LIN {X 0,Y 516.886,Z 94.228,A -85,B 0,C 180,E1 -4924.209,E2 -4924.209} C_VEL
LIN {X 0,Y 516.862,Z 94.224,A -85,B 0,C 180,E1 -4926.776,E2 -4926.776} C_VEL
LIN {X 0,Y 516.942,Z 94.22,A -85,B 0,C 180,E1 -4929.732,E2 -4929.732} C_VEL
LIN {X 0,Y 516.923,Z 94.315,A -85,B 0,C 180,E1 -4932.877,E2 -4932.877} C_VEL
LIN {X 0,Y 518.41,Z 102.009,A -85,B 0,C 180,E1 -4934.268,E2 -4934.268} C_VEL
LIN {X 0,Y 518.118,Z 116.227,A -85,B 0,C 180,E1 -4936.668,E2 -4936.668} C_VEL
LIN {X 0,Y 517.972,Z 120.931,A -85,B 0,C 180,E1 -4937.437,E2 -4937.437} C_VEL
LIN {X 0,Y 520.412,Z 132.652,A -85,B 0,C 180,E1 -4937.694,E2 -4937.694} C_VEL
LIN {X 0,Y 519.711,Z 257.165,A -85,B 0,C 180,E1 -4939.457,E2 -4939.457} C_VEL
LIN {X 0,Y 519.49,Z 271.718,A -85,B 0,C 180,E1 -4939.821,E2 -4939.821} C_VEL
LIN {X 0,Y 519.222,Z 285.007,A -85,B 0,C 180,E1 -4940.308,E2 -4940.308} C_VEL
LIN {X 0,Y 518.835,Z 298.02,A -85,B 0,C 180,E1 -4940.94,E2 -4940.94} C_VEL
LIN {X 0,Y 518.353,Z 311.178,A -85,B 0,C 180,E1 -4941.758,E2 -4941.758} C_VEL
LIN {X 0,Y 517.962,Z 323.367,A -85,B 0,C 180,E1 -4942.706,E2 -4942.706} C_VEL
LIN {X 0,Y 517.606,Z 334.484,A -85,B 0,C 180,E1 -4943.764,E2 -4943.764} C_VEL
LIN {X 0,Y 517.164,Z 344.616,A -85,B 0,C 180,E1 -4944.933,E2 -4944.933} C_VEL
LIN {X 0,Y 516.767,Z 353.015,A -85,B 0,C 180,E1 -4946.101,E2 -4946.101} C_VEL
LIN {X 0,Y 516.612,Z 361.049,A -85,B 0,C 180,E1 -4947.466,E2 -4947.466} C_VEL
LIN {X 0,Y 516.497,Z 367.544,A -85,B 0,C 180,E1 -4948.831,E2 -4948.831} C_VEL
LIN {X 0,Y 516.339,Z 373.334,A -85,B 0,C 180,E1 -4950.39,E2 -4950.39} C_VEL
LIN {X 0,Y 516.219,Z 376.698,A -85,B 0,C 180,E1 -4951.56,E2 -4951.56} C_VEL
LIN {X 0,Y 516.293,Z 379.858,A -85,B 0,C 180,E1 -4953.121,E2 -4953.121} C_VEL
LIN {X 0,Y 516.216,Z 381.664,A -85,B 0,C 180,E1 -4954.686,E2 -4954.686} C_VEL
LIN {X 0,Y 516.295,Z 382.143,A -85,B 0,C 180,E1 -4956.252,E2 -4956.252} C_VEL
LIN {X 0,Y 516.227,Z 381.298,A -85,B 0,C 180,E1 -4957.825,E2 -4957.825} C_VEL
LIN {X 0,Y 516.2,Z 379.096,A -85,B 0,C 180,E1 -4959.403,E2 -4959.403} C_VEL
LIN {X 0,Y 516.363,Z 375.472,A -85,B 0,C 180,E1 -4960.985,E2 -4960.985} C_VEL
LIN {X 0,Y 516.399,Z 370.302,A -85,B 0,C 180,E1 -4962.577,E2 -4962.577} C_VEL
LIN {X 0,Y 516.541,Z 365.25,A -85,B 0,C 180,E1 -4963.775,E2 -4963.775} C_VEL
LIN {X 0,Y 516.733,Z 358.651,A -85,B 0,C 180,E1 -4965.058,E2 -4965.058} C_VEL
LIN {X 0,Y 516.971,Z 350.31,A -85,B 0,C 180,E1 -4966.385,E2 -4966.385} C_VEL
LIN {X 0,Y 517.323,Z 341.381,A -85,B 0,C 180,E1 -4967.554,E2 -4967.554} C_VEL
LIN {X 0,Y 517.693,Z 330.77,A -85,B 0,C 180,E1 -4968.707,E2 -4968.707} C_VEL
LIN {X 0,Y 518.118,Z 319.402,A -85,B 0,C 180,E1 -4969.72,E2 -4969.72} C_VEL
LIN {X 0,Y 518.543,Z 306.72,A -85,B 0,C 180,E1 -4970.633,E2 -4970.633} C_VEL
LIN {X 0,Y 518.93,Z 293.485,A -85,B 0,C 180,E1 -4971.391,E2 -4971.391} C_VEL
LIN {X 0,Y 519.308,Z 279.434,A -85,B 0,C 180,E1 -4972.006,E2 -4972.006} C_VEL
LIN {X 0,Y 519.577,Z 265.737,A -85,B 0,C 180,E1 -4972.439,E2 -4972.439} C_VEL
LIN {X 0,Y 519.75,Z 252.041,A -85,B 0,C 180,E1 -4972.72,E2 -4972.72} C_VEL
LIN {X 0,Y 520.435,Z 132.727,A -85,B 0,C 180,E1 -4974.395,E2 -4974.395} C_VEL
LIN {X 0,Y 517.976,Z 120.735,A -85,B 0,C 180,E1 -4974.681,E2 -4974.681} C_VEL
LIN {X 0,Y 518.432,Z 105.65,A -85,B 0,C 180,E1 -4977.228,E2 -4977.228} C_VEL
LIN {X 0,Y 518.096,Z 100.414,A -85,B 0,C 180,E1 -4978.148,E2 -4978.148} C_VEL
LIN {X 0,Y 516.856,Z 94.228,A -85,B 0,C 180,E1 -4979.309,E2 -4979.309} C_VEL
LIN {X 0,Y 516.865,Z 94.226,A -85,B 0,C 180,E1 -4982.537,E2 -4982.537} C_VEL
LIN {X 0,Y 516.83,Z 94.229,A -85,B 0,C 180,E1 -4985.323,E2 -4985.323} C_VEL
LIN {X 0,Y 516.86,Z 94.224,A -85,B 0,C 180,E1 -4988.718,E2 -4988.718} C_VEL
LIN {X 0,Y 516.832,Z 94.235,A -85,B 0,C 180,E1 -4991.783,E2 -4991.783} C_VEL
LIN {X 0,Y 516.897,Z 94.22,A -85,B 0,C 180,E1 -4995.007,E2 -4995.007} C_VEL
LIN {X 0,Y 516.852,Z 94.225,A -85,B 0,C 180,E1 -4998.407,E2 -4998.407} C_VEL
LIN {X 0,Y 516.872,Z 94.224,A -85,B 0,C 180,E1 -5001.283,E2 -5001.283} C_VEL
LIN {X 0,Y 516.861,Z 94.224,A -85,B 0,C 180,E1 -5004.671,E2 -5004.671} C_VEL
LIN {X 0,Y 516.895,Z 94.223,A -85,B 0,C 180,E1 -5007.457,E2 -5007.457} C_VEL
LIN {X 0,Y 516.904,Z 94.22,A -85,B 0,C 180,E1 -5010.694,E2 -5010.694} C_VEL
LIN {X 0,Y 516.882,Z 94.218,A -85,B 0,C 180,E1 -5013.818,E2 -5013.818} C_VEL
LIN {X 0,Y 516.857,Z 94.23,A -85,B 0,C 180,E1 -5016.776,E2 -5016.776} C_VEL
LIN {X 0,Y 516.938,Z 94.214,A -85,B 0,C 180,E1 -5019.732,E2 -5019.732} C_VEL
LIN {X 0,Y 516.896,Z 94.224,A -85,B 0,C 180,E1 -5022.595,E2 -5022.595} C_VEL
LIN {X 0,Y 516.932,Z 94.215,A -85,B 0,C 180,E1 -5025.03,E2 -5025.03} C_VEL
LIN {X 0,Y 516.967,Z 94.215,A -85,B 0,C 180,E1 -5028.234,E2 -5028.234} C_VEL
LIN {X 0,Y 516.956,Z 94.208,A -85,B 0,C 180,E1 -5031.399,E2 -5031.399} C_VEL
LIN {X 0,Y 517.021,Z 94.205,A -85,B 0,C 180,E1 -5034.54,E2 -5034.54} C_VEL
LIN {X 0,Y 517.081,Z 94.198,A -85,B 0,C 180,E1 -5037.663,E2 -5037.663} C_VEL
LIN {X 0,Y 517.091,Z 94.192,A -85,B 0,C 180,E1 -5040.779,E2 -5040.779} C_VEL
LIN {X 0,Y 516.984,Z 94.208,A -85,B 0,C 180,E1 -5043.117,E2 -5043.117} C_VEL
LIN {X 0,Y 516.977,Z 94.207,A -85,B 0,C 180,E1 -5046.243,E2 -5046.243} C_VEL
LIN {X 0,Y 516.943,Z 94.219,A -85,B 0,C 180,E1 -5049.389,E2 -5049.389} C_VEL
LIN {X 0,Y 516.953,Z 94.215,A -85,B 0,C 180,E1 -5051.807,E2 -5051.807} C_VEL
LIN {X 0,Y 516.944,Z 94.218,A -85,B 0,C 180,E1 -5055.146,E2 -5055.146} C_VEL
LIN {X 0,Y 516.925,Z 94.215,A -85,B 0,C 180,E1 -5058.222,E2 -5058.222} C_VEL
LIN {X 0,Y 516.913,Z 94.217,A -85,B 0,C 180,E1 -5060.701,E2 -5060.701} C_VEL
LIN {X 0,Y 516.903,Z 94.216,A -85,B 0,C 180,E1 -5064.072,E2 -5064.072} C_VEL
LIN {X 0,Y 516.925,Z 94.218,A -85,B 0,C 180,E1 -5066.658,E2 -5066.658} C_VEL
LIN {X 0,Y 516.912,Z 94.217,A -85,B 0,C 180,E1 -5069.524,E2 -5069.524} C_VEL
LIN {X 0,Y 516.899,Z 94.223,A -85,B 0,C 180,E1 -5072.544,E2 -5072.544} C_VEL
LIN {X 0,Y 516.87,Z 94.221,A -85,B 0,C 180,E1 -5075.33,E2 -5075.33} C_VEL
LIN {X 0,Y 516.881,Z 94.222,A -85,B 0,C 180,E1 -5077.943,E2 -5077.943} C_VEL
LIN {X 0,Y 516.885,Z 94.224,A -85,B 0,C 180,E1 -5080.742,E2 -5080.742} C_VEL
LIN {X 0,Y 516.885,Z 94.222,A -85,B 0,C 180,E1 -5082.831,E2 -5082.831} C_VEL
LIN {X 0,Y 516.883,Z 94.225,A -85,B 0,C 180,E1 -5086.097,E2 -5086.097} C_VEL
LIN {X 0,Y 516.916,Z 94.222,A -85,B 0,C 180,E1 -5088.399,E2 -5088.399} C_VEL
LIN {X 0,Y 516.884,Z 94.22,A -85,B 0,C 180,E1 -5091.284,E2 -5091.284} C_VEL
LIN {X 0,Y 516.872,Z 94.226,A -85,B 0,C 180,E1 -5094.22,E2 -5094.22} C_VEL
LIN {X 0,Y 516.896,Z 94.217,A -85,B 0,C 180,E1 -5097.053,E2 -5097.053} C_VEL
LIN {X 0,Y 516.893,Z 94.226,A -85,B 0,C 180,E1 -5099.796,E2 -5099.796} C_VEL
LIN {X 0,Y 516.93,Z 94.219,A -85,B 0,C 180,E1 -5102.467,E2 -5102.467} C_VEL
LIN {X 0,Y 516.957,Z 94.246,A -85,B 0,C 180,E1 -5104.047,E2 -5104.047} C_VEL
LIN {X 0,Y 518.949,Z 103.849,A -85,B 0,C 180,E1 -5105.633,E2 -5105.633} C_VEL
LIN {X 0,Y 518.879,Z 112.01,A -85,B 0,C 180,E1 -5106.872,E2 -5106.872} C_VEL
LIN {X 0,Y 518.251,Z 131.547,A -85,B 0,C 180,E1 -5109.769,E2 -5109.769} C_VEL
LIN {X 0,Y 517.976,Z 142.613,A -85,B 0,C 180,E1 -5111.377,E2 -5111.377} C_VEL
LIN {X 0,Y 520.411,Z 156.781,A -85,B 0,C 180,E1 -5111.67,E2 -5111.67} C_VEL
LIN {X 0,Y 519.606,Z 280.718,A -85,B 0,C 180,E1 -5113.423,E2 -5113.423} C_VEL
LIN {X 0,Y 519.341,Z 295.01,A -85,B 0,C 180,E1 -5113.785,E2 -5113.785} C_VEL
LIN {X 0,Y 519.059,Z 308.626,A -85,B 0,C 180,E1 -5114.288,E2 -5114.288} C_VEL
LIN {X 0,Y 518.678,Z 320.831,A -85,B 0,C 180,E1 -5114.88,E2 -5114.88} C_VEL
LIN {X 0,Y 518.212,Z 333.672,A -85,B 0,C 180,E1 -5115.67,E2 -5115.67} C_VEL
LIN {X 0,Y 517.839,Z 345.351,A -85,B 0,C 180,E1 -5116.56,E2 -5116.56} C_VEL
LIN {X 0,Y 517.487,Z 355.071,A -85,B 0,C 180,E1 -5117.45,E2 -5117.45} C_VEL
LIN {X 0,Y 517.156,Z 365.842,A -85,B 0,C 180,E1 -5118.635,E2 -5118.635} C_VEL
LIN {X 0,Y 516.819,Z 374.735,A -85,B 0,C 180,E1 -5119.818,E2 -5119.818} C_VEL
LIN {X 0,Y 516.608,Z 383.26,A -85,B 0,C 180,E1 -5121.196,E2 -5121.196} C_VEL
LIN {X 0,Y 516.441,Z 390.13,A -85,B 0,C 180,E1 -5122.572,E2 -5122.572} C_VEL
LIN {X 0,Y 516.357,Z 394.866,A -85,B 0,C 180,E1 -5123.749,E2 -5123.749} C_VEL
LIN {X 0,Y 516.303,Z 398.702,A -85,B 0,C 180,E1 -5124.924,E2 -5124.924} C_VEL
LIN {X 0,Y 516.324,Z 401.659,A -85,B 0,C 180,E1 -5126.097,E2 -5126.097} C_VEL
LIN {X 0,Y 516.259,Z 404.364,A -85,B 0,C 180,E1 -5127.659,E2 -5127.659} C_VEL
LIN {X 0,Y 516.156,Z 405.704,A -85,B 0,C 180,E1 -5129.22,E2 -5129.22} C_VEL
LIN {X 0,Y 516.156,Z 405.706,A -85,B 0,C 180,E1 -5130.78,E2 -5130.78} C_VEL
LIN {X 0,Y 516.259,Z 404.371,A -85,B 0,C 180,E1 -5132.34,E2 -5132.34} C_VEL
LIN {X 0,Y 516.324,Z 401.67,A -85,B 0,C 180,E1 -5133.902,E2 -5133.902} C_VEL
LIN {X 0,Y 516.353,Z 397.525,A -85,B 0,C 180,E1 -5135.467,E2 -5135.467} C_VEL
LIN {X 0,Y 516.4,Z 391.816,A -85,B 0,C 180,E1 -5137.035,E2 -5137.035} C_VEL
LIN {X 0,Y 516.565,Z 385.381,A -85,B 0,C 180,E1 -5138.41,E2 -5138.41} C_VEL
LIN {X 0,Y 516.753,Z 377.385,A -85,B 0,C 180,E1 -5139.788,E2 -5139.788} C_VEL
LIN {X 0,Y 517.059,Z 369.025,A -85,B 0,C 180,E1 -5140.97,E2 -5140.97} C_VEL
LIN {X 0,Y 517.408,Z 358.729,A -85,B 0,C 180,E1 -5142.179,E2 -5142.179} C_VEL
LIN {X 0,Y 517.77,Z 347.731,A -85,B 0,C 180,E1 -5143.241,E2 -5143.241} C_VEL
LIN {X 0,Y 518.118,Z 336.563,A -85,B 0,C 180,E1 -5144.132,E2 -5144.132} C_VEL
LIN {X 0,Y 518.536,Z 324.404,A -85,B 0,C 180,E1 -5144.923,E2 -5144.923} C_VEL
LIN {X 0,Y 518.993,Z 310.915,A -85,B 0,C 180,E1 -5145.613,E2 -5145.613} C_VEL
LIN {X 0,Y 519.284,Z 296.756,A -85,B 0,C 180,E1 -5146.16,E2 -5146.16} C_VEL
LIN {X 0,Y 519.595,Z 281.901,A -85,B 0,C 180,E1 -5146.552,E2 -5146.552} C_VEL
LIN {X 0,Y 519.83,Z 251.984,A -85,B 0,C 180,E1 -5146.999,E2 -5146.999} C_VEL
LIN {X 0,Y 520.344,Z 155.931,A -85,B 0,C 180,E1 -5148.345,E2 -5148.345} C_VEL
LIN {X 0,Y 517.993,Z 142.476,A -85,B 0,C 180,E1 -5148.634,E2 -5148.634} C_VEL
LIN {X 0,Y 518.563,Z 120.29,A -85,B 0,C 180,E1 -5151.882,E2 -5151.882} C_VEL
LIN {X 0,Y 519.05,Z 104.898,A -85,B 0,C 180,E1 -5154.163,E2 -5154.163} C_VEL
LIN {X 0,Y 516.961,Z 94.218,A -85,B 0,C 180,E1 -5155.889,E2 -5155.889} C_VEL
LIN {X 0,Y 516.92,Z 94.222,A -85,B 0,C 180,E1 -5158.415,E2 -5158.415} C_VEL
LIN {X 0,Y 516.889,Z 94.221,A -85,B 0,C 180,E1 -5161.109,E2 -5161.109} C_VEL
LIN {X 0,Y 516.908,Z 94.223,A -85,B 0,C 180,E1 -5163.966,E2 -5163.966} C_VEL
LIN {X 0,Y 516.876,Z 94.222,A -85,B 0,C 180,E1 -5166.746,E2 -5166.746} C_VEL
LIN {X 0,Y 516.882,Z 94.225,A -85,B 0,C 180,E1 -5169.721,E2 -5169.721} C_VEL
LIN {X 0,Y 516.914,Z 94.223,A -85,B 0,C 180,E1 -5171.775,E2 -5171.775} C_VEL
LIN {X 0,Y 516.922,Z 94.215,A -85,B 0,C 180,E1 -5175.01,E2 -5175.01} C_VEL
LIN {X 0,Y 516.915,Z 94.217,A -85,B 0,C 180,E1 -5178.398,E2 -5178.398} C_VEL
LIN {X 0,Y 516.879,Z 94.225,A -85,B 0,C 180,E1 -5181.284,E2 -5181.284} C_VEL
LIN {X 0,Y 516.87,Z 94.222,A -85,B 0,C 180,E1 -5184.22,E2 -5184.22} C_VEL
LIN {X 0,Y 516.895,Z 94.222,A -85,B 0,C 180,E1 -5187.053,E2 -5187.053} C_VEL
LIN {X 0,Y 516.891,Z 94.221,A -85,B 0,C 180,E1 -5189.796,E2 -5189.796} C_VEL
LIN {X 0,Y 516.925,Z 94.215,A -85,B 0,C 180,E1 -5192.467,E2 -5192.467} C_VEL
LIN {X 0,Y 516.908,Z 94.225,A -85,B 0,C 180,E1 -5195.072,E2 -5195.072} C_VEL
LIN {X 0,Y 516.884,Z 94.222,A -85,B 0,C 180,E1 -5198.462,E2 -5198.462} C_VEL
LIN {X 0,Y 516.901,Z 94.227,A -85,B 0,C 180,E1 -5200.955,E2 -5200.955} C_VEL
LIN {X 0,Y 516.912,Z 94.218,A -85,B 0,C 180,E1 -5203.41,E2 -5203.41} C_VEL
LIN {X 0,Y 516.895,Z 94.218,A -85,B 0,C 180,E1 -5205.834,E2 -5205.834} C_VEL
LIN {X 0,Y 516.965,Z 94.212,A -85,B 0,C 180,E1 -5208.234,E2 -5208.234} C_VEL
LIN {X 0,Y 516.967,Z 94.21,A -85,B 0,C 180,E1 -5211.4,E2 -5211.4} C_VEL
LIN {X 0,Y 517.008,Z 94.205,A -85,B 0,C 180,E1 -5213.757,E2 -5213.757} C_VEL
LIN {X 0,Y 517.082,Z 94.196,A -85,B 0,C 180,E1 -5217.663,E2 -5217.663} C_VEL
LIN {X 0,Y 517.092,Z 94.196,A -85,B 0,C 180,E1 -5220.779,E2 -5220.779} C_VEL
LIN {X 0,Y 517.011,Z 94.204,A -85,B 0,C 180,E1 -5223.117,E2 -5223.117} C_VEL
LIN {X 0,Y 516.988,Z 94.214,A -85,B 0,C 180,E1 -5226.244,E2 -5226.244} C_VEL
LIN {X 0,Y 516.968,Z 94.211,A -85,B 0,C 180,E1 -5228.601,E2 -5228.601} C_VEL
LIN {X 0,Y 516.952,Z 94.219,A -85,B 0,C 180,E1 -5231.807,E2 -5231.807} C_VEL
LIN {X 0,Y 516.944,Z 94.213,A -85,B 0,C 180,E1 -5235.147,E2 -5235.147} C_VEL
LIN {X 0,Y 516.912,Z 94.218,A -85,B 0,C 180,E1 -5238.223,E2 -5238.223} C_VEL
LIN {X 0,Y 516.912,Z 94.216,A -85,B 0,C 180,E1 -5240.702,E2 -5240.702} C_VEL
LIN {X 0,Y 516.891,Z 94.221,A -85,B 0,C 180,E1 -5244.073,E2 -5244.073} C_VEL
LIN {X 0,Y 516.925,Z 94.215,A -85,B 0,C 180,E1 -5246.658,E2 -5246.658} C_VEL
LIN {X 0,Y 516.908,Z 94.223,A -85,B 0,C 180,E1 -5249.524,E2 -5249.524} C_VEL
LIN {X 0,Y 516.894,Z 94.219,A -85,B 0,C 180,E1 -5252.543,E2 -5252.543} C_VEL
LIN {X 0,Y 516.865,Z 94.228,A -85,B 0,C 180,E1 -5255.33,E2 -5255.33} C_VEL
LIN {X 0,Y 516.879,Z 94.22,A -85,B 0,C 180,E1 -5257.943,E2 -5257.943} C_VEL
LIN {X 0,Y 516.883,Z 94.225,A -85,B 0,C 180,E1 -5260.742,E2 -5260.742} C_VEL
LIN {X 0,Y 516.883,Z 94.228,A -85,B 0,C 180,E1 -5262.832,E2 -5262.832} C_VEL
LIN {X 0,Y 516.896,Z 94.224,A -85,B 0,C 180,E1 -5265.007,E2 -5265.007} C_VEL
LIN {X 0,Y 516.911,Z 94.221,A -85,B 0,C 180,E1 -5268.4,E2 -5268.4} C_VEL
LIN {X 0,Y 516.882,Z 94.224,A -85,B 0,C 180,E1 -5270.287,E2 -5270.287} C_VEL
LIN {X 0,Y 516.207,Z 94.309,A -85,B 0,C 180,E1 -5270.937,E2 -5270.937} C_VEL
LIN {X 0,Y 513.349,Z 94.662,A -85,B 0,C 180,E1 -5271.993,E2 -5271.993} C_VEL
LIN {X 0,Y 510.935,Z 94.966,A -85,B 0,C 180,E1 -5272.843,E2 -5272.843} C_VEL
LIN {X 0,Y 509.895,Z 95.091,A -85,B 0,C 180,E1 -5273.499,E2 -5273.499} C_VEL
LIN {X 0,Y 509.808,Z 95.102,A -85,B 0,C 180,E1 -5273.722,E2 -5273.722} C_VEL
LIN {X 0,Y 509.86,Z 95.102,A -85,B 0,C 180,E1 -5276.539,E2 -5276.539} C_VEL
LIN {X 0,Y 509.847,Z 95.096,A -85,B 0,C 180,E1 -5279.335,E2 -5279.335} C_VEL
LIN {X 0,Y 509.847,Z 95.102,A -85,B 0,C 180,E1 -5282.052,E2 -5282.052} C_VEL
LIN {X 0,Y 509.817,Z 95.102,A -85,B 0,C 180,E1 -5284.701,E2 -5284.701} C_VEL
LIN {X 0,Y 509.829,Z 95.1,A -85,B 0,C 180,E1 -5287.458,E2 -5287.458} C_VEL
LIN {X 0,Y 509.919,Z 95.096,A -85,B 0,C 180,E1 -5289.845,E2 -5289.845} C_VEL
LIN {X 0,Y 509.892,Z 95.19,A -85,B 0,C 180,E1 -5292.685,E2 -5292.685} C_VEL
LIN {X 0,Y 511.532,Z 104.027,A -85,B 0,C 180,E1 -5294.299,E2 -5294.299} C_VEL
LIN {X 0,Y 511.03,Z 120.993,A -85,B 0,C 180,E1 -5297.18,E2 -5297.18} C_VEL
LIN {X 0,Y 513.74,Z 134.085,A -85,B 0,C 180,E1 -5297.47,E2 -5297.47} C_VEL
LIN {X 0,Y 512.923,Z 257.73,A -85,B 0,C 180,E1 -5299.241,E2 -5299.241} C_VEL
LIN {X 0,Y 512.673,Z 272.139,A -85,B 0,C 180,E1 -5299.61,E2 -5299.61} C_VEL
LIN {X 0,Y 512.372,Z 285.921,A -85,B 0,C 180,E1 -5300.128,E2 -5300.128} C_VEL
LIN {X 0,Y 511.921,Z 299.648,A -85,B 0,C 180,E1 -5300.817,E2 -5300.817} C_VEL
LIN {X 0,Y 511.442,Z 312.046,A -85,B 0,C 180,E1 -5301.611,E2 -5301.611} C_VEL
LIN {X 0,Y 511.025,Z 324.435,A -85,B 0,C 180,E1 -5302.6,E2 -5302.6} C_VEL
LIN {X 0,Y 510.626,Z 335.443,A -85,B 0,C 180,E1 -5303.679,E2 -5303.679} C_VEL
LIN {X 0,Y 510.151,Z 345.407,A -85,B 0,C 180,E1 -5304.863,E2 -5304.863} C_VEL
LIN {X 0,Y 509.725,Z 353.706,A -85,B 0,C 180,E1 -5306.047,E2 -5306.047} C_VEL
LIN {X 0,Y 509.557,Z 361.633,A -85,B 0,C 180,E1 -5307.431,E2 -5307.431} C_VEL
LIN {X 0,Y 509.413,Z 368.046,A -85,B 0,C 180,E1 -5308.814,E2 -5308.814} C_VEL
LIN {X 0,Y 509.262,Z 373.758,A -85,B 0,C 180,E1 -5310.395,E2 -5310.395} C_VEL
LIN {X 0,Y 509.138,Z 377.054,A -85,B 0,C 180,E1 -5311.582,E2 -5311.582} C_VEL
LIN {X 0,Y 509.207,Z 380.139,A -85,B 0,C 180,E1 -5313.165,E2 -5313.165} C_VEL
LIN {X 0,Y 509.131,Z 381.877,A -85,B 0,C 180,E1 -5314.751,E2 -5314.751} C_VEL
LIN {X 0,Y 509.221,Z 382.271,A -85,B 0,C 180,E1 -5316.429,E2 -5316.429} C_VEL
LIN {X 0,Y 509.142,Z 381.376,A -85,B 0,C 180,E1 -5317.934,E2 -5317.934} C_VEL
LIN {X 0,Y 509.114,Z 379.104,A -85,B 0,C 180,E1 -5319.535,E2 -5319.535} C_VEL
LIN {X 0,Y 509.298,Z 375.407,A -85,B 0,C 180,E1 -5321.139,E2 -5321.139} C_VEL
LIN {X 0,Y 509.363,Z 370.155,A -85,B 0,C 180,E1 -5322.754,E2 -5322.754} C_VEL
LIN {X 0,Y 509.495,Z 365.022,A -85,B 0,C 180,E1 -5323.969,E2 -5323.969} C_VEL
LIN {X 0,Y 509.754,Z 357.657,A -85,B 0,C 180,E1 -5325.391,E2 -5325.391} C_VEL
LIN {X 0,Y 510.054,Z 348.445,A -85,B 0,C 180,E1 -5326.82,E2 -5326.82} C_VEL
LIN {X 0,Y 510.414,Z 338.458,A -85,B 0,C 180,E1 -5328.077,E2 -5328.077} C_VEL
LIN {X 0,Y 510.865,Z 327.876,A -85,B 0,C 180,E1 -5329.175,E2 -5329.175} C_VEL
LIN {X 0,Y 511.32,Z 315.823,A -85,B 0,C 180,E1 -5330.201,E2 -5330.201} C_VEL
LIN {X 0,Y 511.771,Z 304.056,A -85,B 0,C 180,E1 -5331.014,E2 -5331.014} C_VEL
LIN {X 0,Y 512.189,Z 291.84,A -85,B 0,C 180,E1 -5331.692,E2 -5331.692} C_VEL
LIN {X 0,Y 512.525,Z 278.694,A -85,B 0,C 180,E1 -5332.26,E2 -5332.26} C_VEL
LIN {X 0,Y 512.776,Z 264.818,A -85,B 0,C 180,E1 -5332.695,E2 -5332.695} C_VEL
LIN {X 0,Y 512.975,Z 251.108,A -85,B 0,C 180,E1 -5332.967,E2 -5332.967} C_VEL
LIN {X 0,Y 513.774,Z 134.042,A -85,B 0,C 180,E1 -5334.631,E2 -5334.631} C_VEL
LIN {X 0,Y 511.065,Z 120.93,A -85,B 0,C 180,E1 -5334.944,E2 -5334.944} C_VEL
LIN {X 0,Y 511.57,Z 105.313,A -85,B 0,C 180,E1 -5337.624,E2 -5337.624} C_VEL
LIN {X 0,Y 510.327,Z 97.623,A -85,B 0,C 180,E1 -5339.042,E2 -5339.042} C_VEL
LIN {X 0,Y 509.808,Z 95.107,A -85,B 0,C 180,E1 -5339.538,E2 -5339.538} C_VEL
LIN {X 0,Y 509.833,Z 95.103,A -85,B 0,C 180,E1 -5342.521,E2 -5342.521} C_VEL
LIN {X 0,Y 509.791,Z 95.106,A -85,B 0,C 180,E1 -5345.381,E2 -5345.381} C_VEL
LIN {X 0,Y 509.809,Z 95.105,A -85,B 0,C 180,E1 -5348.342,E2 -5348.342} C_VEL
LIN {X 0,Y 509.784,Z 95.111,A -85,B 0,C 180,E1 -5351.433,E2 -5351.433} C_VEL
LIN {X 0,Y 509.836,Z 95.099,A -85,B 0,C 180,E1 -5354.67,E2 -5354.67} C_VEL
LIN {X 0,Y 509.79,Z 95.112,A -85,B 0,C 180,E1 -5357.505,E2 -5357.505} C_VEL
LIN {X 0,Y 509.831,Z 95.094,A -85,B 0,C 180,E1 -5360.646,E2 -5360.646} C_VEL
LIN {X 0,Y 509.804,Z 95.105,A -85,B 0,C 180,E1 -5363.645,E2 -5363.645} C_VEL
LIN {X 0,Y 509.84,Z 95.099,A -85,B 0,C 180,E1 -5366.537,E2 -5366.537} C_VEL
LIN {X 0,Y 509.834,Z 95.102,A -85,B 0,C 180,E1 -5369.333,E2 -5369.333} C_VEL
LIN {X 0,Y 509.834,Z 95.099,A -85,B 0,C 180,E1 -5372.051,E2 -5372.051} C_VEL
LIN {X 0,Y 509.802,Z 95.106,A -85,B 0,C 180,E1 -5374.7,E2 -5374.7} C_VEL
LIN {X 0,Y 509.825,Z 95.098,A -85,B 0,C 180,E1 -5377.459,E2 -5377.459} C_VEL
LIN {X 0,Y 509.916,Z 95.089,A -85,B 0,C 180,E1 -5379.844,E2 -5379.844} C_VEL
LIN {X 0,Y 509.864,Z 95.096,A -85,B 0,C 180,E1 -5383.174,E2 -5383.174} C_VEL
LIN {X 0,Y 509.847,Z 95.096,A -85,B 0,C 180,E1 -5385.633,E2 -5385.633} C_VEL
LIN {X 0,Y 509.913,Z 95.091,A -85,B 0,C 180,E1 -5388.874,E2 -5388.874} C_VEL
LIN {X 0,Y 509.922,Z 95.09,A -85,B 0,C 180,E1 -5392.078,E2 -5392.078} C_VEL
LIN {X 0,Y 509.972,Z 95.084,A -85,B 0,C 180,E1 -5394.464,E2 -5394.464} C_VEL
LIN {X 0,Y 510.051,Z 95.073,A -85,B 0,C 180,E1 -5397.631,E2 -5397.631} C_VEL
LIN {X 0,Y 510.062,Z 95.067,A -85,B 0,C 180,E1 -5400.789,E2 -5400.789} C_VEL
LIN {X 0,Y 509.928,Z 95.087,A -85,B 0,C 180,E1 -5403.16,E2 -5403.16} C_VEL
LIN {X 0,Y 509.924,Z 95.085,A -85,B 0,C 180,E1 -5406.33,E2 -5406.33} C_VEL
LIN {X 0,Y 509.911,Z 95.089,A -85,B 0,C 180,E1 -5408.72,E2 -5408.72} C_VEL
LIN {X 0,Y 509.905,Z 95.091,A -85,B 0,C 180,E1 -5411.932,E2 -5411.932} C_VEL
LIN {X 0,Y 509.895,Z 95.097,A -85,B 0,C 180,E1 -5415.242,E2 -5415.242} C_VEL
LIN {X 0,Y 509.883,Z 95.093,A -85,B 0,C 180,E1 -5417.998,E2 -5417.998} C_VEL
LIN {X 0,Y 509.851,Z 95.099,A -85,B 0,C 180,E1 -5421.002,E2 -5421.002} C_VEL
LIN {X 0,Y 509.865,Z 95.094,A -85,B 0,C 180,E1 -5424.426,E2 -5424.426} C_VEL
LIN {X 0,Y 509.885,Z 95.098,A -85,B 0,C 180,E1 -5427.056,E2 -5427.056} C_VEL
LIN {X 0,Y 509.858,Z 95.095,A -85,B 0,C 180,E1 -5429.751,E2 -5429.751} C_VEL
LIN {X 0,Y 509.876,Z 95.099,A -85,B 0,C 180,E1 -5432.774,E2 -5432.774} C_VEL
LIN {X 0,Y 509.828,Z 95.098,A -85,B 0,C 180,E1 -5435.579,E2 -5435.579} C_VEL
LIN {X 0,Y 509.85,Z 95.103,A -85,B 0,C 180,E1 -5438.338,E2 -5438.338} C_VEL
LIN {X 0,Y 509.857,Z 95.095,A -85,B 0,C 180,E1 -5441.425,E2 -5441.425} C_VEL
LIN {X 0,Y 509.84,Z 95.1,A -85,B 0,C 180,E1 -5444.67,E2 -5444.67} C_VEL
LIN {X 0,Y 509.835,Z 95.1,A -85,B 0,C 180,E1 -5447.51,E2 -5447.51} C_VEL
LIN {X 0,Y 509.848,Z 95.097,A -85,B 0,C 180,E1 -5450.648,E2 -5450.648} C_VEL
LIN {X 0,Y 509.826,Z 95.103,A -85,B 0,C 180,E1 -5453.647,E2 -5453.647} C_VEL
LIN {X 0,Y 509.86,Z 95.093,A -85,B 0,C 180,E1 -5456.539,E2 -5456.539} C_VEL
LIN {X 0,Y 509.847,Z 95.1,A -85,B 0,C 180,E1 -5459.334,E2 -5459.334} C_VEL
LIN {X 0,Y 509.895,Z 95.098,A -85,B 0,C 180,E1 -5462.055,E2 -5462.055} C_VEL
LIN {X 0,Y 509.949,Z 95.299,A -85,B 0,C 180,E1 -5463.831,E2 -5463.831} C_VEL
LIN {X 0,Y 512.172,Z 106.4,A -85,B 0,C 180,E1 -5465.691,E2 -5465.691} C_VEL
LIN {X 0,Y 511.65,Z 123.095,A -85,B 0,C 180,E1 -5468.231,E2 -5468.231} C_VEL
LIN {X 0,Y 511.065,Z 142.619,A -85,B 0,C 180,E1 -5471.112,E2 -5471.112} C_VEL
LIN {X 0,Y 513.686,Z 157.572,A -85,B 0,C 180,E1 -5471.431,E2 -5471.431} C_VEL
LIN {X 0,Y 512.807,Z 280.587,A -85,B 0,C 180,E1 -5473.196,E2 -5473.196} C_VEL
LIN {X 0,Y 512.533,Z 294.614,A -85,B 0,C 180,E1 -5473.555,E2 -5473.555} C_VEL
LIN {X 0,Y 512.202,Z 308.464,A -85,B 0,C 180,E1 -5474.072,E2 -5474.072} C_VEL
LIN {X 0,Y 511.727,Z 322.43,A -85,B 0,C 180,E1 -5474.772,E2 -5474.772} C_VEL
LIN {X 0,Y 511.247,Z 334.93,A -85,B 0,C 180,E1 -5475.572,E2 -5475.572} C_VEL
LIN {X 0,Y 510.847,Z 346.358,A -85,B 0,C 180,E1 -5476.474,E2 -5476.474} C_VEL
LIN {X 0,Y 510.453,Z 356.862,A -85,B 0,C 180,E1 -5477.476,E2 -5477.476} C_VEL
LIN {X 0,Y 510.114,Z 367.308,A -85,B 0,C 180,E1 -5478.678,E2 -5478.678} C_VEL
LIN {X 0,Y 509.758,Z 375.928,A -85,B 0,C 180,E1 -5479.876,E2 -5479.876} C_VEL
LIN {X 0,Y 509.521,Z 384.185,A -85,B 0,C 180,E1 -5481.273,E2 -5481.273} C_VEL
LIN {X 0,Y 509.365,Z 389.964,A -85,B 0,C 180,E1 -5482.468,E2 -5482.468} C_VEL
LIN {X 0,Y 509.263,Z 394.7,A -85,B 0,C 180,E1 -5483.661,E2 -5483.661} C_VEL
LIN {X 0,Y 509.232,Z 398.538,A -85,B 0,C 180,E1 -5484.853,E2 -5484.853} C_VEL
LIN {X 0,Y 509.216,Z 401.494,A -85,B 0,C 180,E1 -5486.043,E2 -5486.043} C_VEL
LIN {X 0,Y 509.188,Z 404.201,A -85,B 0,C 180,E1 -5487.627,E2 -5487.627} C_VEL
LIN {X 0,Y 509.07,Z 405.541,A -85,B 0,C 180,E1 -5489.209,E2 -5489.209} C_VEL
LIN {X 0,Y 509.07,Z 405.543,A -85,B 0,C 180,E1 -5490.791,E2 -5490.791} C_VEL
LIN {X 0,Y 509.188,Z 404.209,A -85,B 0,C 180,E1 -5492.373,E2 -5492.373} C_VEL
LIN {X 0,Y 509.216,Z 401.507,A -85,B 0,C 180,E1 -5493.957,E2 -5493.957} C_VEL
LIN {X 0,Y 509.267,Z 397.362,A -85,B 0,C 180,E1 -5495.543,E2 -5495.543} C_VEL
LIN {X 0,Y 509.325,Z 391.652,A -85,B 0,C 180,E1 -5497.134,E2 -5497.134} C_VEL
LIN {X 0,Y 509.508,Z 385.217,A -85,B 0,C 180,E1 -5498.527,E2 -5498.527} C_VEL
LIN {X 0,Y 509.708,Z 377.221,A -85,B 0,C 180,E1 -5499.925,E2 -5499.925} C_VEL
LIN {X 0,Y 510.036,Z 368.86,A -85,B 0,C 180,E1 -5501.123,E2 -5501.123} C_VEL
LIN {X 0,Y 510.391,Z 358.154,A -85,B 0,C 180,E1 -5502.394,E2 -5502.394} C_VEL
LIN {X 0,Y 510.817,Z 347.565,A -85,B 0,C 180,E1 -5503.425,E2 -5503.425} C_VEL
LIN {X 0,Y 511.204,Z 336.397,A -85,B 0,C 180,E1 -5504.327,E2 -5504.327} C_VEL
LIN {X 0,Y 511.644,Z 324.236,A -85,B 0,C 180,E1 -5505.128,E2 -5505.128} C_VEL
LIN {X 0,Y 512.148,Z 310.745,A -85,B 0,C 180,E1 -5505.827,E2 -5505.827} C_VEL
LIN {X 0,Y 512.46,Z 296.743,A -85,B 0,C 180,E1 -5506.376,E2 -5506.376} C_VEL
LIN {X 0,Y 512.791,Z 282.839,A -85,B 0,C 180,E1 -5506.753,E2 -5506.753} C_VEL
LIN {X 0,Y 513.005,Z 262.477,A -85,B 0,C 180,E1 -5507.079,E2 -5507.079} C_VEL
LIN {X 0,Y 513.559,Z 156.679,A -85,B 0,C 180,E1 -5508.581,E2 -5508.581} C_VEL
LIN {X 0,Y 511.044,Z 142.305,A -85,B 0,C 180,E1 -5508.893,E2 -5508.893} C_VEL
LIN {X 0,Y 511.639,Z 121.473,A -85,B 0,C 180,E1 -5511.982,E2 -5511.982} C_VEL
LIN {X 0,Y 512.11,Z 105.965,A -85,B 0,C 180,E1 -5514.312,E2 -5514.312} C_VEL
LIN {X 0,Y 509.909,Z 95.097,A -85,B 0,C 180,E1 -5516.116,E2 -5516.116} C_VEL
LIN {X 0,Y 509.877,Z 95.098,A -85,B 0,C 180,E1 -5518.844,E2 -5518.844} C_VEL
LIN {X 0,Y 509.82,Z 95.103,A -85,B 0,C 180,E1 -5521.59,E2 -5521.59} C_VEL
LIN {X 0,Y 509.847,Z 95.101,A -85,B 0,C 180,E1 -5524.414,E2 -5524.414} C_VEL
LIN {X 0,Y 509.817,Z 95.101,A -85,B 0,C 180,E1 -5527.341,E2 -5527.341} C_VEL
LIN {X 0,Y 509.838,Z 95.1,A -85,B 0,C 180,E1 -5530.382,E2 -5530.382} C_VEL
LIN {X 0,Y 509.824,Z 95.1,A -85,B 0,C 180,E1 -5533.062,E2 -5533.062} C_VEL
LIN {X 0,Y 509.831,Z 95.107,A -85,B 0,C 180,E1 -5535.792,E2 -5535.792} C_VEL
LIN {X 0,Y 509.856,Z 95.095,A -85,B 0,C 180,E1 -5538.575,E2 -5538.575} C_VEL
LIN {X 0,Y 509.85,Z 95.102,A -85,B 0,C 180,E1 -5541.786,E2 -5541.786} C_VEL
LIN {X 0,Y 509.829,Z 95.099,A -85,B 0,C 180,E1 -5544.622,E2 -5544.622} C_VEL
LIN {X 0,Y 509.862,Z 95.102,A -85,B 0,C 180,E1 -5547.481,E2 -5547.481} C_VEL
LIN {X 0,Y 509.857,Z 95.095,A -85,B 0,C 180,E1 -5550.274,E2 -5550.274} C_VEL
LIN {X 0,Y 509.883,Z 95.097,A -85,B 0,C 180,E1 -5552.944,E2 -5552.944} C_VEL
LIN {X 0,Y 509.864,Z 95.097,A -85,B 0,C 180,E1 -5555.574,E2 -5555.574} C_VEL
LIN {X 0,Y 509.849,Z 95.105,A -85,B 0,C 180,E1 -5558.998,E2 -5558.998} C_VEL
LIN {X 0,Y 509.881,Z 95.092,A -85,B 0,C 180,E1 -5562.002,E2 -5562.002} C_VEL
LIN {X 0,Y 509.909,Z 95.098,A -85,B 0,C 180,E1 -5564.819,E2 -5564.819} C_VEL
LIN {X 0,Y 509.9,Z 95.091,A -85,B 0,C 180,E1 -5568.124,E2 -5568.124} C_VEL
LIN {X 0,Y 509.913,Z 95.089,A -85,B 0,C 180,E1 -5571.28,E2 -5571.28} C_VEL
LIN {X 0,Y 509.958,Z 95.083,A -85,B 0,C 180,E1 -5573.67,E2 -5573.67} C_VEL
LIN {X 0,Y 510.053,Z 95.071,A -85,B 0,C 180,E1 -5577.631,E2 -5577.631} C_VEL
LIN {X 0,Y 510.062,Z 95.072,A -85,B 0,C 180,E1 -5580.79,E2 -5580.79} C_VEL
LIN {X 0,Y 509.953,Z 95.083,A -85,B 0,C 180,E1 -5583.16,E2 -5583.16} C_VEL
LIN {X 0,Y 509.936,Z 95.091,A -85,B 0,C 180,E1 -5586.33,E2 -5586.33} C_VEL
LIN {X 0,Y 509.914,Z 95.089,A -85,B 0,C 180,E1 -5588.72,E2 -5588.72} C_VEL
LIN {X 0,Y 509.904,Z 95.098,A -85,B 0,C 180,E1 -5591.932,E2 -5591.932} C_VEL
LIN {X 0,Y 509.894,Z 95.092,A -85,B 0,C 180,E1 -5595.242,E2 -5595.242} C_VEL
LIN {X 0,Y 509.857,Z 95.096,A -85,B 0,C 180,E1 -5598.484,E2 -5598.484} C_VEL
LIN {X 0,Y 509.85,Z 95.097,A -85,B 0,C 180,E1 -5601.002,E2 -5601.002} C_VEL
LIN {X 0,Y 509.822,Z 95.108,A -85,B 0,C 180,E1 -5603.564,E2 -5603.564} C_VEL
LIN {X 0,Y 509.911,Z 95.088,A -85,B 0,C 180,E1 -5606.379,E2 -5606.379} C_VEL
LIN {X 0,Y 509.872,Z 95.095,A -85,B 0,C 180,E1 -5608.845,E2 -5608.845} C_VEL
LIN {X 0,Y 509.819,Z 95.104,A -85,B 0,C 180,E1 -5611.591,E2 -5611.591} C_VEL
LIN {X 0,Y 509.838,Z 95.098,A -85,B 0,C 180,E1 -5614.415,E2 -5614.415} C_VEL
LIN {X 0,Y 509.816,Z 95.105,A -85,B 0,C 180,E1 -5617.341,E2 -5617.341} C_VEL
LIN {X 0,Y 509.838,Z 95.099,A -85,B 0,C 180,E1 -5620.383,E2 -5620.383} C_VEL
LIN {X 0,Y 509.823,Z 95.105,A -85,B 0,C 180,E1 -5623.062,E2 -5623.062} C_VEL
LIN {X 0,Y 509.822,Z 95.099,A -85,B 0,C 180,E1 -5625.794,E2 -5625.794} C_VEL
LIN {X 0,Y 509.853,Z 95.103,A -85,B 0,C 180,E1 -5628.575,E2 -5628.575} C_VEL
LIN {X 0,Y 509.851,Z 95.096,A -85,B 0,C 180,E1 -5631.787,E2 -5631.787} C_VEL
LIN {X 0,Y 509.808,Z 95.102,A -85,B 0,C 180,E1 -5633.722,E2 -5633.722} C_VEL
LIN {X 0,Y 509.148,Z 95.19,A -85,B 0,C 180,E1 -5634.382,E2 -5634.382} C_VEL
LIN {X 0,Y 506.343,Z 95.537,A -85,B 0,C 180,E1 -5635.454,E2 -5635.454} C_VEL
LIN {X 0,Y 503.957,Z 95.837,A -85,B 0,C 180,E1 -5636.318,E2 -5636.318} C_VEL
LIN {X 0,Y 502.909,Z 95.963,A -85,B 0,C 180,E1 -5636.984,E2 -5636.984} C_VEL
LIN {X 0,Y 502.811,Z 95.973,A -85,B 0,C 180,E1 -5637.21,E2 -5637.21} C_VEL
LIN {X 0,Y 502.817,Z 95.977,A -85,B 0,C 180,E1 -5640.065,E2 -5640.065} C_VEL
LIN {X 0,Y 502.814,Z 95.973,A -85,B 0,C 180,E1 -5643.431,E2 -5643.431} C_VEL
LIN {X 0,Y 502.775,Z 95.986,A -85,B 0,C 180,E1 -5646.086,E2 -5646.086} C_VEL
LIN {X 0,Y 502.786,Z 95.979,A -85,B 0,C 180,E1 -5648.689,E2 -5648.689} C_VEL
LIN {X 0,Y 502.825,Z 95.976,A -85,B 0,C 180,E1 -5651.248,E2 -5651.248} C_VEL
LIN {X 0,Y 502.84,Z 96.053,A -85,B 0,C 180,E1 -5652.486,E2 -5652.486} C_VEL
LIN {X 0,Y 504.48,Z 104.187,A -85,B 0,C 180,E1 -5653.999,E2 -5653.999} C_VEL
LIN {X 0,Y 504.411,Z 112.677,A -85,B 0,C 180,E1 -5655.476,E2 -5655.476} C_VEL
LIN {X 0,Y 504.119,Z 121.081,A -85,B 0,C 180,E1 -5656.914,E2 -5656.914} C_VEL
LIN {X 0,Y 506.985,Z 134.716,A -85,B 0,C 180,E1 -5657.229,E2 -5657.229} C_VEL
LIN {X 0,Y 506.121,Z 258.055,A -85,B 0,C 180,E1 -5659.018,E2 -5659.018} C_VEL
LIN {X 0,Y 505.867,Z 272.423,A -85,B 0,C 180,E1 -5659.393,E2 -5659.393} C_VEL
LIN {X 0,Y 505.575,Z 285.633,A -85,B 0,C 180,E1 -5659.892,E2 -5659.892} C_VEL
LIN {X 0,Y 505.152,Z 297.732,A -85,B 0,C 180,E1 -5660.491,E2 -5660.491} C_VEL
LIN {X 0,Y 504.642,Z 310.529,A -85,B 0,C 180,E1 -5661.295,E2 -5661.295} C_VEL
LIN {X 0,Y 504.136,Z 323.154,A -85,B 0,C 180,E1 -5662.289,E2 -5662.289} C_VEL
LIN {X 0,Y 503.704,Z 334.508,A -85,B 0,C 180,E1 -5663.39,E2 -5663.39} C_VEL
LIN {X 0,Y 503.226,Z 344.7,A -85,B 0,C 180,E1 -5664.591,E2 -5664.591} C_VEL
LIN {X 0,Y 502.756,Z 353.141,A -85,B 0,C 180,E1 -5665.791,E2 -5665.791} C_VEL
LIN {X 0,Y 502.561,Z 361.223,A -85,B 0,C 180,E1 -5667.195,E2 -5667.195} C_VEL
LIN {X 0,Y 502.262,Z 366.905,A -85,B 0,C 180,E1 -5668.396,E2 -5668.396} C_VEL
LIN {X 0,Y 502.253,Z 371.563,A -85,B 0,C 180,E1 -5669.599,E2 -5669.599} C_VEL
LIN {X 0,Y 502.146,Z 376.417,A -85,B 0,C 180,E1 -5671.203,E2 -5671.203} C_VEL
LIN {X 0,Y 502.123,Z 379.083,A -85,B 0,C 180,E1 -5672.407,E2 -5672.407} C_VEL
LIN {X 0,Y 502.09,Z 381.421,A -85,B 0,C 180,E1 -5674.013,E2 -5674.013} C_VEL
LIN {X 0,Y 502.106,Z 382.427,A -85,B 0,C 180,E1 -5675.623,E2 -5675.623} C_VEL
LIN {X 0,Y 502.107,Z 382.111,A -85,B 0,C 180,E1 -5677.237,E2 -5677.237} C_VEL
LIN {X 0,Y 502.05,Z 380.456,A -85,B 0,C 180,E1 -5678.858,E2 -5678.858} C_VEL
LIN {X 0,Y 502.143,Z 377.412,A -85,B 0,C 180,E1 -5680.483,E2 -5680.483} C_VEL
LIN {X 0,Y 502.224,Z 372.881,A -85,B 0,C 180,E1 -5682.117,E2 -5682.117} C_VEL
LIN {X 0,Y 502.35,Z 368.35,A -85,B 0,C 180,E1 -5683.347,E2 -5683.347} C_VEL
LIN {X 0,Y 502.528,Z 362.803,A -85,B 0,C 180,E1 -5684.58,E2 -5684.58} C_VEL
LIN {X 0,Y 502.824,Z 354.836,A -85,B 0,C 180,E1 -5686.024,E2 -5686.024} C_VEL
LIN {X 0,Y 503.152,Z 346.456,A -85,B 0,C 180,E1 -5687.267,E2 -5687.267} C_VEL
LIN {X 0,Y 503.584,Z 336.682,A -85,B 0,C 180,E1 -5688.468,E2 -5688.468} C_VEL
LIN {X 0,Y 504.036,Z 326.048,A -85,B 0,C 180,E1 -5689.551,E2 -5689.551} C_VEL
LIN {X 0,Y 504.491,Z 313.925,A -85,B 0,C 180,E1 -5690.564,E2 -5690.564} C_VEL
LIN {X 0,Y 505.049,Z 300.986,A -85,B 0,C 180,E1 -5691.425,E2 -5691.425} C_VEL
LIN {X 0,Y 505.48,Z 288.11,A -85,B 0,C 180,E1 -5692.103,E2 -5692.103} C_VEL
LIN {X 0,Y 505.829,Z 273.538,A -85,B 0,C 180,E1 -5692.679,E2 -5692.679} C_VEL
LIN {X 0,Y 506.098,Z 259.231,A -85,B 0,C 180,E1 -5693.065,E2 -5693.065} C_VEL
LIN {X 0,Y 506.416,Z 225.137,A -85,B 0,C 180,E1 -5693.584,E2 -5693.584} C_VEL
LIN {X 0,Y 506.935,Z 134.242,A -85,B 0,C 180,E1 -5694.901,E2 -5694.901} C_VEL
LIN {X 0,Y 504.198,Z 121.109,A -85,B 0,C 180,E1 -5695.222,E2 -5695.222} C_VEL
LIN {X 0,Y 504.652,Z 106.262,A -85,B 0,C 180,E1 -5697.81,E2 -5697.81} C_VEL
LIN {X 0,Y 503.097,Z 97.452,A -85,B 0,C 180,E1 -5699.471,E2 -5699.471} C_VEL
LIN {X 0,Y 502.749,Z 95.988,A -85,B 0,C 180,E1 -5699.769,E2 -5699.769} C_VEL
LIN {X 0,Y 502.757,Z 95.989,A -85,B 0,C 180,E1 -5702.087,E2 -5702.087} C_VEL
LIN {X 0,Y 502.755,Z 95.981,A -85,B 0,C 180,E1 -5704.969,E2 -5704.969} C_VEL
LIN {X 0,Y 502.755,Z 95.983,A -85,B 0,C 180,E1 -5708.48,E2 -5708.48} C_VEL
LIN {X 0,Y 502.75,Z 95.983,A -85,B 0,C 180,E1 -5711.073,E2 -5711.073} C_VEL
LIN {X 0,Y 502.779,Z 95.978,A -85,B 0,C 180,E1 -5714.529,E2 -5714.529} C_VEL
LIN {X 0,Y 502.767,Z 95.983,A -85,B 0,C 180,E1 -5717.857,E2 -5717.857} C_VEL
LIN {X 0,Y 502.783,Z 95.975,A -85,B 0,C 180,E1 -5721.022,E2 -5721.022} C_VEL
LIN {X 0,Y 502.769,Z 95.978,A -85,B 0,C 180,E1 -5724.17,E2 -5724.17} C_VEL
LIN {X 0,Y 502.832,Z 95.976,A -85,B 0,C 180,E1 -5726.994,E2 -5726.994} C_VEL
LIN {X 0,Y 502.811,Z 95.972,A -85,B 0,C 180,E1 -5730.066,E2 -5730.066} C_VEL
LIN {X 0,Y 502.784,Z 95.976,A -85,B 0,C 180,E1 -5733.429,E2 -5733.429} C_VEL
LIN {X 0,Y 502.766,Z 95.98,A -85,B 0,C 180,E1 -5736.085,E2 -5736.085} C_VEL
LIN {X 0,Y 502.781,Z 95.982,A -85,B 0,C 180,E1 -5738.689,E2 -5738.689} C_VEL
LIN {X 0,Y 502.823,Z 95.97,A -85,B 0,C 180,E1 -5741.248,E2 -5741.248} C_VEL
LIN {X 0,Y 502.85,Z 95.975,A -85,B 0,C 180,E1 -5744.6,E2 -5744.6} C_VEL
LIN {X 0,Y 502.878,Z 95.968,A -85,B 0,C 180,E1 -5748.039,E2 -5748.039} C_VEL
LIN {X 0,Y 502.864,Z 95.962,A -85,B 0,C 180,E1 -5751.156,E2 -5751.156} C_VEL
LIN {X 0,Y 502.926,Z 95.963,A -85,B 0,C 180,E1 -5754.386,E2 -5754.386} C_VEL
LIN {X 0,Y 503.02,Z 95.948,A -85,B 0,C 180,E1 -5757.598,E2 -5757.598} C_VEL
LIN {X 0,Y 503.011,Z 95.945,A -85,B 0,C 180,E1 -5760.8,E2 -5760.8} C_VEL
LIN {X 0,Y 503.021,Z 95.949,A -85,B 0,C 180,E1 -5762.402,E2 -5762.402} C_VEL
LIN {X 0,Y 502.919,Z 95.965,A -85,B 0,C 180,E1 -5765.614,E2 -5765.614} C_VEL
LIN {X 0,Y 502.869,Z 95.967,A -85,B 0,C 180,E1 -5768.843,E2 -5768.843} C_VEL
LIN {X 0,Y 502.846,Z 95.969,A -85,B 0,C 180,E1 -5772.102,E2 -5772.102} C_VEL
LIN {X 0,Y 502.849,Z 95.972,A -85,B 0,C 180,E1 -5775.4,E2 -5775.4} C_VEL
LIN {X 0,Y 502.842,Z 95.969,A -85,B 0,C 180,E1 -5778.12,E2 -5778.12} C_VEL
LIN {X 0,Y 502.83,Z 95.969,A -85,B 0,C 180,E1 -5780.536,E2 -5780.536} C_VEL
LIN {X 0,Y 502.791,Z 95.983,A -85,B 0,C 180,E1 -5783.04,E2 -5783.04} C_VEL
LIN {X 0,Y 502.841,Z 95.969,A -85,B 0,C 180,E1 -5785.675,E2 -5785.675} C_VEL
LIN {X 0,Y 502.841,Z 95.971,A -85,B 0,C 180,E1 -5788.373,E2 -5788.373} C_VEL
LIN {X 0,Y 502.795,Z 95.975,A -85,B 0,C 180,E1 -5791.499,E2 -5791.499} C_VEL
LIN {X 0,Y 502.806,Z 95.975,A -85,B 0,C 180,E1 -5793.994,E2 -5793.994} C_VEL
LIN {X 0,Y 502.778,Z 95.979,A -85,B 0,C 180,E1 -5797.178,E2 -5797.178} C_VEL
LIN {X 0,Y 502.788,Z 95.973,A -85,B 0,C 180,E1 -5800.015,E2 -5800.015} C_VEL
LIN {X 0,Y 502.803,Z 95.98,A -85,B 0,C 180,E1 -5802.199,E2 -5802.199} C_VEL
LIN {X 0,Y 502.786,Z 95.975,A -85,B 0,C 180,E1 -5805.47,E2 -5805.47} C_VEL
LIN {X 0,Y 502.821,Z 95.973,A -85,B 0,C 180,E1 -5808.934,E2 -5808.934} C_VEL
LIN {X 0,Y 502.795,Z 95.981,A -85,B 0,C 180,E1 -5812.046,E2 -5812.046} C_VEL
LIN {X 0,Y 502.8,Z 95.974,A -85,B 0,C 180,E1 -5815.034,E2 -5815.034} C_VEL
LIN {X 0,Y 502.784,Z 95.981,A -85,B 0,C 180,E1 -5817.915,E2 -5817.915} C_VEL
LIN {X 0,Y 502.826,Z 95.974,A -85,B 0,C 180,E1 -5820.712,E2 -5820.712} C_VEL
LIN {X 0,Y 502.892,Z 96.055,A -85,B 0,C 180,E1 -5823.557,E2 -5823.557} C_VEL
LIN {X 0,Y 505.274,Z 107.77,A -85,B 0,C 180,E1 -5825.556,E2 -5825.556} C_VEL
LIN {X 0,Y 504.806,Z 121.659,A -85,B 0,C 180,E1 -5827.705,E2 -5827.705} C_VEL
LIN {X 0,Y 504.173,Z 141.123,A -85,B 0,C 180,E1 -5830.666,E2 -5830.666} C_VEL
LIN {X 0,Y 504.081,Z 142.166,A -85,B 0,C 180,E1 -5830.821,E2 -5830.821} C_VEL
LIN {X 0,Y 506.983,Z 159.199,A -85,B 0,C 180,E1 -5831.193,E2 -5831.193} C_VEL
LIN {X 0,Y 506.066,Z 279.499,A -85,B 0,C 180,E1 -5832.94,E2 -5832.94} C_VEL
LIN {X 0,Y 505.752,Z 293.808,A -85,B 0,C 180,E1 -5833.301,E2 -5833.301} C_VEL
LIN {X 0,Y 505.388,Z 307.22,A -85,B 0,C 180,E1 -5833.798,E2 -5833.798} C_VEL
LIN {X 0,Y 504.927,Z 320.561,A -85,B 0,C 180,E1 -5834.458,E2 -5834.458} C_VEL
LIN {X 0,Y 504.413,Z 333.373,A -85,B 0,C 180,E1 -5835.269,E2 -5835.269} C_VEL
LIN {X 0,Y 503.923,Z 345.029,A -85,B 0,C 180,E1 -5836.182,E2 -5836.182} C_VEL
LIN {X 0,Y 503.477,Z 355.817,A -85,B 0,C 180,E1 -5837.207,E2 -5837.207} C_VEL
LIN {X 0,Y 503.11,Z 365.558,A -85,B 0,C 180,E1 -5838.32,E2 -5838.32} C_VEL
LIN {X 0,Y 502.794,Z 374.4,A -85,B 0,C 180,E1 -5839.53,E2 -5839.53} C_VEL
LIN {X 0,Y 502.487,Z 382.925,A -85,B 0,C 180,E1 -5840.947,E2 -5840.947} C_VEL
LIN {X 0,Y 502.289,Z 389.797,A -85,B 0,C 180,E1 -5842.361,E2 -5842.361} C_VEL
LIN {X 0,Y 502.165,Z 395.308,A -85,B 0,C 180,E1 -5843.789,E2 -5843.789} C_VEL
LIN {X 0,Y 502.101,Z 399.443,A -85,B 0,C 180,E1 -5845.182,E2 -5845.182} C_VEL
LIN {X 0,Y 502.112,Z 402.858,A -85,B 0,C 180,E1 -5846.79,E2 -5846.79} C_VEL
LIN {X 0,Y 502.033,Z 404.877,A -85,B 0,C 180,E1 -5848.395,E2 -5848.395} C_VEL
LIN {X 0,Y 501.981,Z 405.547,A -85,B 0,C 180,E1 -5850,E2 -5850} C_VEL
LIN {X 0,Y 502.033,Z 404.882,A -85,B 0,C 180,E1 -5851.604,E2 -5851.604} C_VEL
LIN {X 0,Y 502.112,Z 402.869,A -85,B 0,C 180,E1 -5853.209,E2 -5853.209} C_VEL
LIN {X 0,Y 502.101,Z 399.458,A -85,B 0,C 180,E1 -5854.817,E2 -5854.817} C_VEL
LIN {X 0,Y 502.168,Z 395.308,A -85,B 0,C 180,E1 -5856.214,E2 -5856.214} C_VEL
LIN {X 0,Y 502.289,Z 389.814,A -85,B 0,C 180,E1 -5857.638,E2 -5857.638} C_VEL
LIN {X 0,Y 502.487,Z 382.948,A -85,B 0,C 180,E1 -5859.053,E2 -5859.053} C_VEL
LIN {X 0,Y 502.794,Z 374.426,A -85,B 0,C 180,E1 -5860.469,E2 -5860.469} C_VEL
LIN {X 0,Y 503.15,Z 364.397,A -85,B 0,C 180,E1 -5861.827,E2 -5861.827} C_VEL
LIN {X 0,Y 503.518,Z 354.758,A -85,B 0,C 180,E1 -5862.904,E2 -5862.904} C_VEL
LIN {X 0,Y 503.967,Z 343.855,A -85,B 0,C 180,E1 -5863.919,E2 -5863.919} C_VEL
LIN {X 0,Y 504.473,Z 331.918,A -85,B 0,C 180,E1 -5864.832,E2 -5864.832} C_VEL
LIN {X 0,Y 504.962,Z 318.689,A -85,B 0,C 180,E1 -5865.644,E2 -5865.644} C_VEL
LIN {X 0,Y 505.427,Z 304.918,A -85,B 0,C 180,E1 -5866.291,E2 -5866.291} C_VEL
LIN {X 0,Y 505.778,Z 291.06,A -85,B 0,C 180,E1 -5866.77,E2 -5866.77} C_VEL
LIN {X 0,Y 506.045,Z 277.302,A -85,B 0,C 180,E1 -5867.087,E2 -5867.087} C_VEL
LIN {X 0,Y 506.81,Z 157.593,A -85,B 0,C 180,E1 -5868.814,E2 -5868.814} C_VEL
LIN {X 0,Y 504.077,Z 142.217,A -85,B 0,C 180,E1 -5869.143,E2 -5869.143} C_VEL
LIN {X 0,Y 504.694,Z 122.635,A -85,B 0,C 180,E1 -5872.085,E2 -5872.085} C_VEL
LIN {X 0,Y 505.219,Z 108.529,A -85,B 0,C 180,E1 -5874.228,E2 -5874.228} C_VEL
LIN {X 0,Y 503.942,Z 101.014,A -85,B 0,C 180,E1 -5875.455,E2 -5875.455} C_VEL
LIN {X 0,Y 502.867,Z 95.974,A -85,B 0,C 180,E1 -5876.339,E2 -5876.339} C_VEL
LIN {X 0,Y 502.825,Z 95.974,A -85,B 0,C 180,E1 -5879.288,E2 -5879.288} C_VEL
LIN {X 0,Y 502.783,Z 95.985,A -85,B 0,C 180,E1 -5882.084,E2 -5882.084} C_VEL
LIN {X 0,Y 502.799,Z 95.975,A -85,B 0,C 180,E1 -5884.966,E2 -5884.966} C_VEL
LIN {X 0,Y 502.793,Z 95.983,A -85,B 0,C 180,E1 -5887.954,E2 -5887.954} C_VEL
LIN {X 0,Y 502.82,Z 95.972,A -85,B 0,C 180,E1 -5891.066,E2 -5891.066} C_VEL
LIN {X 0,Y 502.8,Z 95.975,A -85,B 0,C 180,E1 -5894.532,E2 -5894.532} C_VEL
LIN {X 0,Y 502.829,Z 95.977,A -85,B 0,C 180,E1 -5897.864,E2 -5897.864} C_VEL
LIN {X 0,Y 502.8,Z 95.976,A -85,B 0,C 180,E1 -5901.024,E2 -5901.024} C_VEL
LIN {X 0,Y 502.774,Z 95.978,A -85,B 0,C 180,E1 -5904.169,E2 -5904.169} C_VEL
LIN {X 0,Y 502.832,Z 95.973,A -85,B 0,C 180,E1 -5906.993,E2 -5906.993} C_VEL
LIN {X 0,Y 502.814,Z 95.973,A -85,B 0,C 180,E1 -5910.065,E2 -5910.065} C_VEL
LIN {X 0,Y 502.831,Z 95.971,A -85,B 0,C 180,E1 -5912.533,E2 -5912.533} C_VEL
LIN {X 0,Y 502.826,Z 95.977,A -85,B 0,C 180,E1 -5915.299,E2 -5915.299} C_VEL
LIN {X 0,Y 502.779,Z 95.977,A -85,B 0,C 180,E1 -5917.826,E2 -5917.826} C_VEL
LIN {X 0,Y 502.823,Z 95.973,A -85,B 0,C 180,E1 -5920.4,E2 -5920.4} C_VEL
LIN {X 0,Y 502.829,Z 95.979,A -85,B 0,C 180,E1 -5922.932,E2 -5922.932} C_VEL
LIN {X 0,Y 502.844,Z 95.97,A -85,B 0,C 180,E1 -5925.429,E2 -5925.429} C_VEL
LIN {X 0,Y 502.876,Z 95.973,A -85,B 0,C 180,E1 -5928.717,E2 -5928.717} C_VEL
LIN {X 0,Y 502.901,Z 95.963,A -85,B 0,C 180,E1 -5931.967,E2 -5931.967} C_VEL
LIN {X 0,Y 502.934,Z 95.965,A -85,B 0,C 180,E1 -5934.387,E2 -5934.387} C_VEL
LIN {X 0,Y 503.023,Z 95.947,A -85,B 0,C 180,E1 -5937.598,E2 -5937.598} C_VEL
LIN {X 0,Y 503.027,Z 95.95,A -85,B 0,C 180,E1 -5940,E2 -5940} C_VEL
LIN {X 0,Y 503.023,Z 95.953,A -85,B 0,C 180,E1 -5942.402,E2 -5942.402} C_VEL
LIN {X 0,Y 502.926,Z 95.961,A -85,B 0,C 180,E1 -5945.614,E2 -5945.614} C_VEL
LIN {X 0,Y 502.873,Z 95.965,A -85,B 0,C 180,E1 -5948.843,E2 -5948.843} C_VEL
LIN {X 0,Y 502.846,Z 95.974,A -85,B 0,C 180,E1 -5952.102,E2 -5952.102} C_VEL
LIN {X 0,Y 502.848,Z 95.972,A -85,B 0,C 180,E1 -5955.4,E2 -5955.4} C_VEL
LIN {X 0,Y 502.822,Z 95.972,A -85,B 0,C 180,E1 -5958.752,E2 -5958.752} C_VEL
LIN {X 0,Y 502.783,Z 95.981,A -85,B 0,C 180,E1 -5961.311,E2 -5961.311} C_VEL
LIN {X 0,Y 502.775,Z 95.981,A -85,B 0,C 180,E1 -5963.915,E2 -5963.915} C_VEL
LIN {X 0,Y 502.864,Z 95.966,A -85,B 0,C 180,E1 -5966.566,E2 -5966.566} C_VEL
LIN {X 0,Y 502.822,Z 95.98,A -85,B 0,C 180,E1 -5969.288,E2 -5969.288} C_VEL
LIN {X 0,Y 502.782,Z 95.977,A -85,B 0,C 180,E1 -5972.085,E2 -5972.085} C_VEL
LIN {X 0,Y 502.795,Z 95.981,A -85,B 0,C 180,E1 -5974.966,E2 -5974.966} C_VEL
LIN {X 0,Y 502.792,Z 95.975,A -85,B 0,C 180,E1 -5977.954,E2 -5977.954} C_VEL
LIN {X 0,Y 502.82,Z 95.979,A -85,B 0,C 180,E1 -5981.066,E2 -5981.066} C_VEL
LIN {X 0,Y 502.786,Z 95.98,A -85,B 0,C 180,E1 -5984.53,E2 -5984.53} C_VEL
LIN {X 0,Y 502.795,Z 95.975,A -85,B 0,C 180,E1 -5987.861,E2 -5987.861} C_VEL
LIN {X 0,Y 502.802,Z 95.977,A -85,B 0,C 180,E1 -5991.024,E2 -5991.024} C_VEL
LIN {X 0,Y 502.772,Z 95.982,A -85,B 0,C 180,E1 -5994.17,E2 -5994.17} C_VEL
LIN {X 0,Y 502.811,Z 95.973,A -85,B 0,C 180,E1 -5997.21,E2 -5997.21} C_VEL
LIN {X 0,Y 502.11,Z 96.064,A -85,B 0,C 180,E1 -5997.878,E2 -5997.878} C_VEL
LIN {X 0,Y 499.249,Z 96.42,A -85,B 0,C 180,E1 -5998.964,E2 -5998.964} C_VEL
LIN {X 0,Y 496.85,Z 96.721,A -85,B 0,C 180,E1 -5999.839,E2 -5999.839} C_VEL
LIN {X 0,Y 495.823,Z 96.849,A -85,B 0,C 180,E1 -6000.515,E2 -6000.515} C_VEL
LIN {X 0,Y 495.738,Z 96.856,A -85,B 0,C 180,E1 -6000.743,E2 -6000.743} C_VEL
LIN {X 0,Y 495.739,Z 96.859,A -85,B 0,C 180,E1 -6003.929,E2 -6003.929} C_VEL
LIN {X 0,Y 495.761,Z 96.851,A -85,B 0,C 180,E1 -6007.14,E2 -6007.14} C_VEL
LIN {X 0,Y 495.772,Z 96.858,A -85,B 0,C 180,E1 -6010.11,E2 -6010.11} C_VEL
LIN {X 0,Y 495.814,Z 97.054,A -85,B 0,C 180,E1 -6012.31,E2 -6012.31} C_VEL
LIN {X 0,Y 497.599,Z 106.215,A -85,B 0,C 180,E1 -6014.032,E2 -6014.032} C_VEL
LIN {X 0,Y 497.354,Z 118.034,A -85,B 0,C 180,E1 -6016.1,E2 -6016.1} C_VEL
LIN {X 0,Y 497.225,Z 121.229,A -85,B 0,C 180,E1 -6016.652,E2 -6016.652} C_VEL
LIN {X 0,Y 500.273,Z 136.962,A -85,B 0,C 180,E1 -6017.011,E2 -6017.011} C_VEL
LIN {X 0,Y 499.316,Z 258.194,A -85,B 0,C 180,E1 -6018.79,E2 -6018.79} C_VEL
LIN {X 0,Y 499.028,Z 272.583,A -85,B 0,C 180,E1 -6019.168,E2 -6019.168} C_VEL
LIN {X 0,Y 498.729,Z 286.353,A -85,B 0,C 180,E1 -6019.701,E2 -6019.701} C_VEL
LIN {X 0,Y 498.243,Z 299.217,A -85,B 0,C 180,E1 -6020.357,E2 -6020.357} C_VEL
LIN {X 0,Y 497.707,Z 311.691,A -85,B 0,C 180,E1 -6021.167,E2 -6021.167} C_VEL
LIN {X 0,Y 497.226,Z 323.056,A -85,B 0,C 180,E1 -6022.079,E2 -6022.079} C_VEL
LIN {X 0,Y 496.797,Z 333.506,A -85,B 0,C 180,E1 -6023.094,E2 -6023.094} C_VEL
LIN {X 0,Y 496.282,Z 343.904,A -85,B 0,C 180,E1 -6024.311,E2 -6024.311} C_VEL
LIN {X 0,Y 495.841,Z 352.503,A -85,B 0,C 180,E1 -6025.529,E2 -6025.529} C_VEL
LIN {X 0,Y 495.543,Z 360.765,A -85,B 0,C 180,E1 -6026.951,E2 -6026.951} C_VEL
LIN {X 0,Y 495.186,Z 367.439,A -85,B 0,C 180,E1 -6028.374,E2 -6028.374} C_VEL
LIN {X 0,Y 495.041,Z 373.377,A -85,B 0,C 180,E1 -6030,E2 -6030} C_VEL
LIN {X 0,Y 494.985,Z 377.752,A -85,B 0,C 180,E1 -6031.627,E2 -6031.627} C_VEL
LIN {X 0,Y 495.041,Z 380.7,A -85,B 0,C 180,E1 -6033.256,E2 -6033.256} C_VEL
LIN {X 0,Y 494.972,Z 382.303,A -85,B 0,C 180,E1 -6034.887,E2 -6034.887} C_VEL
LIN {X 0,Y 495.053,Z 382.58,A -85,B 0,C 180,E1 -6036.521,E2 -6036.521} C_VEL
LIN {X 0,Y 494.954,Z 381.532,A -85,B 0,C 180,E1 -6038.163,E2 -6038.163} C_VEL
LIN {X 0,Y 494.974,Z 379.122,A -85,B 0,C 180,E1 -6039.81,E2 -6039.81} C_VEL
LIN {X 0,Y 495.137,Z 375.277,A -85,B 0,C 180,E1 -6041.462,E2 -6041.462} C_VEL
LIN {X 0,Y 495.252,Z 369.805,A -85,B 0,C 180,E1 -6043.124,E2 -6043.124} C_VEL
LIN {X 0,Y 495.469,Z 363.568,A -85,B 0,C 180,E1 -6044.583,E2 -6044.583} C_VEL
LIN {X 0,Y 495.765,Z 355.741,A -85,B 0,C 180,E1 -6046.048,E2 -6046.048} C_VEL
LIN {X 0,Y 496.112,Z 347.527,A -85,B 0,C 180,E1 -6047.307,E2 -6047.307} C_VEL
LIN {X 0,Y 496.555,Z 338.114,A -85,B 0,C 180,E1 -6048.506,E2 -6048.506} C_VEL
LIN {X 0,Y 497.046,Z 327.546,A -85,B 0,C 180,E1 -6049.622,E2 -6049.622} C_VEL
LIN {X 0,Y 497.572,Z 315.364,A -85,B 0,C 180,E1 -6050.678,E2 -6050.678} C_VEL
LIN {X 0,Y 498.097,Z 303.313,A -85,B 0,C 180,E1 -6051.522,E2 -6051.522} C_VEL
LIN {X 0,Y 498.612,Z 290.007,A -85,B 0,C 180,E1 -6052.26,E2 -6052.26} C_VEL
LIN {X 0,Y 499.036,Z 276.077,A -85,B 0,C 180,E1 -6052.841,E2 -6052.841} C_VEL
LIN {X 0,Y 499.321,Z 262.14,A -85,B 0,C 180,E1 -6053.251,E2 -6053.251} C_VEL
LIN {X 0,Y 499.503,Z 244.181,A -85,B 0,C 180,E1 -6053.566,E2 -6053.566} C_VEL
LIN {X 0,Y 500.275,Z 135.288,A -85,B 0,C 180,E1 -6055.163,E2 -6055.163} C_VEL
LIN {X 0,Y 497.308,Z 121.201,A -85,B 0,C 180,E1 -6055.527,E2 -6055.527} C_VEL
LIN {X 0,Y 497.773,Z 108.496,A -85,B 0,C 180,E1 -6057.77,E2 -6057.77} C_VEL
LIN {X 0,Y 496.863,Z 102.231,A -85,B 0,C 180,E1 -6058.954,E2 -6058.954} C_VEL
LIN {X 0,Y 495.717,Z 96.865,A -85,B 0,C 180,E1 -6060.03,E2 -6060.03} C_VEL
LIN {X 0,Y 495.726,Z 96.86,A -85,B 0,C 180,E1 -6062.598,E2 -6062.598} C_VEL
LIN {X 0,Y 495.717,Z 96.861,A -85,B 0,C 180,E1 -6065.54,E2 -6065.54} C_VEL
LIN {X 0,Y 495.73,Z 96.857,A -85,B 0,C 180,E1 -6068.763,E2 -6068.763} C_VEL
LIN {X 0,Y 495.701,Z 96.867,A -85,B 0,C 180,E1 -6071.787,E2 -6071.787} C_VEL
LIN {X 0,Y 495.736,Z 96.858,A -85,B 0,C 180,E1 -6075.141,E2 -6075.141} C_VEL
LIN {X 0,Y 495.724,Z 96.857,A -85,B 0,C 180,E1 -6078.215,E2 -6078.215} C_VEL
LIN {X 0,Y 495.74,Z 96.854,A -85,B 0,C 180,E1 -6081.235,E2 -6081.235} C_VEL
LIN {X 0,Y 495.743,Z 96.853,A -85,B 0,C 180,E1 -6084.462,E2 -6084.462} C_VEL
LIN {X 0,Y 495.767,Z 96.856,A -85,B 0,C 180,E1 -6087.405,E2 -6087.405} C_VEL
LIN {X 0,Y 495.758,Z 96.85,A -85,B 0,C 180,E1 -6090.253,E2 -6090.253} C_VEL
LIN {X 0,Y 495.74,Z 96.855,A -85,B 0,C 180,E1 -6093.27,E2 -6093.27} C_VEL
LIN {X 0,Y 495.739,Z 96.861,A -85,B 0,C 180,E1 -6096.612,E2 -6096.612} C_VEL
LIN {X 0,Y 495.78,Z 96.851,A -85,B 0,C 180,E1 -6099.324,E2 -6099.324} C_VEL
LIN {X 0,Y 495.78,Z 96.847,A -85,B 0,C 180,E1 -6101.828,E2 -6101.828} C_VEL
LIN {X 0,Y 495.825,Z 96.85,A -85,B 0,C 180,E1 -6104.549,E2 -6104.549} C_VEL
LIN {X 0,Y 495.83,Z 96.845,A -85,B 0,C 180,E1 -6107.965,E2 -6107.965} C_VEL
LIN {X 0,Y 495.834,Z 96.838,A -85,B 0,C 180,E1 -6111.03,E2 -6111.03} C_VEL
LIN {X 0,Y 495.881,Z 96.842,A -85,B 0,C 180,E1 -6114.306,E2 -6114.306} C_VEL
LIN {X 0,Y 495.988,Z 96.824,A -85,B 0,C 180,E1 -6117.564,E2 -6117.564} C_VEL
LIN {X 0,Y 495.962,Z 96.823,A -85,B 0,C 180,E1 -6120.812,E2 -6120.812} C_VEL
LIN {X 0,Y 495.989,Z 96.824,A -85,B 0,C 180,E1 -6122.436,E2 -6122.436} C_VEL
LIN {X 0,Y 495.874,Z 96.841,A -85,B 0,C 180,E1 -6125.694,E2 -6125.694} C_VEL
LIN {X 0,Y 495.838,Z 96.843,A -85,B 0,C 180,E1 -6128.97,E2 -6128.97} C_VEL
LIN {X 0,Y 495.829,Z 96.844,A -85,B 0,C 180,E1 -6132.035,E2 -6132.035} C_VEL
LIN {X 0,Y 495.825,Z 96.846,A -85,B 0,C 180,E1 -6135.451,E2 -6135.451} C_VEL
LIN {X 0,Y 495.808,Z 96.845,A -85,B 0,C 180,E1 -6138.247,E2 -6138.247} C_VEL
LIN {X 0,Y 495.775,Z 96.85,A -85,B 0,C 180,E1 -6140.756,E2 -6140.756} C_VEL
LIN {X 0,Y 495.748,Z 96.856,A -85,B 0,C 180,E1 -6143.387,E2 -6143.387} C_VEL
LIN {X 0,Y 495.791,Z 96.847,A -85,B 0,C 180,E1 -6146.068,E2 -6146.068} C_VEL
LIN {X 0,Y 495.773,Z 96.854,A -85,B 0,C 180,E1 -6148.815,E2 -6148.815} C_VEL
LIN {X 0,Y 495.757,Z 96.851,A -85,B 0,C 180,E1 -6151.725,E2 -6151.725} C_VEL
LIN {X 0,Y 495.772,Z 96.856,A -85,B 0,C 180,E1 -6154.694,E2 -6154.694} C_VEL
LIN {X 0,Y 495.729,Z 96.856,A -85,B 0,C 180,E1 -6157.562,E2 -6157.562} C_VEL
LIN {X 0,Y 495.767,Z 96.854,A -85,B 0,C 180,E1 -6160.7,E2 -6160.7} C_VEL
LIN {X 0,Y 495.729,Z 96.859,A -85,B 0,C 180,E1 -6164.002,E2 -6164.002} C_VEL
LIN {X 0,Y 495.727,Z 96.857,A -85,B 0,C 180,E1 -6167.117,E2 -6167.117} C_VEL
LIN {X 0,Y 495.76,Z 96.857,A -85,B 0,C 180,E1 -6169.953,E2 -6169.953} C_VEL
LIN {X 0,Y 495.729,Z 96.857,A -85,B 0,C 180,E1 -6172.553,E2 -6172.553} C_VEL
LIN {X 0,Y 495.779,Z 96.851,A -85,B 0,C 180,E1 -6175.457,E2 -6175.457} C_VEL
LIN {X 0,Y 495.757,Z 96.854,A -85,B 0,C 180,E1 -6178.364,E2 -6178.364} C_VEL
LIN {X 0,Y 495.789,Z 96.855,A -85,B 0,C 180,E1 -6181.507,E2 -6181.507} C_VEL
LIN {X 0,Y 495.839,Z 96.97,A -85,B 0,C 180,E1 -6183.298,E2 -6183.298} C_VEL
LIN {X 0,Y 498.384,Z 109.15,A -85,B 0,C 180,E1 -6185.418,E2 -6185.418} C_VEL
LIN {X 0,Y 498.109,Z 118.855,A -85,B 0,C 180,E1 -6186.95,E2 -6186.95} C_VEL
LIN {X 0,Y 497.308,Z 138.282,A -85,B 0,C 180,E1 -6189.958,E2 -6189.958} C_VEL
LIN {X 0,Y 497.236,Z 141.917,A -85,B 0,C 180,E1 -6190.518,E2 -6190.518} C_VEL
LIN {X 0,Y 500.301,Z 159.133,A -85,B 0,C 180,E1 -6190.92,E2 -6190.92} C_VEL
LIN {X 0,Y 499.296,Z 279.866,A -85,B 0,C 180,E1 -6192.701,E2 -6192.701} C_VEL
LIN {X 0,Y 498.969,Z 293.68,A -85,B 0,C 180,E1 -6193.057,E2 -6193.057} C_VEL
LIN {X 0,Y 498.551,Z 307.266,A -85,B 0,C 180,E1 -6193.569,E2 -6193.569} C_VEL
LIN {X 0,Y 498.084,Z 320.55,A -85,B 0,C 180,E1 -6194.239,E2 -6194.239} C_VEL
LIN {X 0,Y 497.508,Z 333.318,A -85,B 0,C 180,E1 -6195.06,E2 -6195.06} C_VEL
LIN {X 0,Y 496.998,Z 344.945,A -85,B 0,C 180,E1 -6195.986,E2 -6195.986} C_VEL
LIN {X 0,Y 496.474,Z 356.585,A -85,B 0,C 180,E1 -6197.117,E2 -6197.117} C_VEL
LIN {X 0,Y 496.082,Z 367.204,A -85,B 0,C 180,E1 -6198.378,E2 -6198.378} C_VEL
LIN {X 0,Y 495.69,Z 375.612,A -85,B 0,C 180,E1 -6199.585,E2 -6199.585} C_VEL
LIN {X 0,Y 495.389,Z 383.858,A -85,B 0,C 180,E1 -6201.022,E2 -6201.022} C_VEL
LIN {X 0,Y 495.207,Z 389.635,A -85,B 0,C 180,E1 -6202.251,E2 -6202.251} C_VEL
LIN {X 0,Y 495.066,Z 395.556,A -85,B 0,C 180,E1 -6203.819,E2 -6203.819} C_VEL
LIN {X 0,Y 495.027,Z 399.279,A -85,B 0,C 180,E1 -6205.113,E2 -6205.113} C_VEL
LIN {X 0,Y 495.032,Z 402.694,A -85,B 0,C 180,E1 -6206.744,E2 -6206.744} C_VEL
LIN {X 0,Y 494.959,Z 404.714,A -85,B 0,C 180,E1 -6208.373,E2 -6208.373} C_VEL
LIN {X 0,Y 494.898,Z 405.384,A -85,B 0,C 180,E1 -6210,E2 -6210} C_VEL
LIN {X 0,Y 494.959,Z 404.72,A -85,B 0,C 180,E1 -6211.627,E2 -6211.627} C_VEL
LIN {X 0,Y 495.032,Z 402.707,A -85,B 0,C 180,E1 -6213.255,E2 -6213.255} C_VEL
LIN {X 0,Y 495.027,Z 399.295,A -85,B 0,C 180,E1 -6214.886,E2 -6214.886} C_VEL
LIN {X 0,Y 495.105,Z 394.384,A -85,B 0,C 180,E1 -6216.52,E2 -6216.52} C_VEL
LIN {X 0,Y 495.276,Z 387.829,A -85,B 0,C 180,E1 -6218.158,E2 -6218.158} C_VEL
LIN {X 0,Y 495.508,Z 380.534,A -85,B 0,C 180,E1 -6219.593,E2 -6219.593} C_VEL
LIN {X 0,Y 495.877,Z 371.493,A -85,B 0,C 180,E1 -6221.03,E2 -6221.03} C_VEL
LIN {X 0,Y 496.218,Z 362,A -85,B 0,C 180,E1 -6222.266,E2 -6222.266} C_VEL
LIN {X 0,Y 496.7,Z 351.491,A -85,B 0,C 180,E1 -6223.397,E2 -6223.397} C_VEL
LIN {X 0,Y 497.202,Z 339.882,A -85,B 0,C 180,E1 -6224.426,E2 -6224.426} C_VEL
LIN {X 0,Y 497.781,Z 326.996,A -85,B 0,C 180,E1 -6225.35,E2 -6225.35} C_VEL
LIN {X 0,Y 498.282,Z 314.391,A -85,B 0,C 180,E1 -6226.069,E2 -6226.069} C_VEL
LIN {X 0,Y 498.682,Z 300.88,A -85,B 0,C 180,E1 -6226.665,E2 -6226.665} C_VEL
LIN {X 0,Y 499.078,Z 287.323,A -85,B 0,C 180,E1 -6227.095,E2 -6227.095} C_VEL
LIN {X 0,Y 499.303,Z 273.54,A -85,B 0,C 180,E1 -6227.377,E2 -6227.377} C_VEL
LIN {X 0,Y 500.147,Z 159.464,A -85,B 0,C 180,E1 -6229.032,E2 -6229.032} C_VEL
LIN {X 0,Y 497.142,Z 142.071,A -85,B 0,C 180,E1 -6229.404,E2 -6229.404} C_VEL
LIN {X 0,Y 497.784,Z 122.369,A -85,B 0,C 180,E1 -6232.408,E2 -6232.408} C_VEL
LIN {X 0,Y 498.314,Z 109.666,A -85,B 0,C 180,E1 -6234.364,E2 -6234.364} C_VEL
LIN {X 0,Y 496.677,Z 101.024,A -85,B 0,C 180,E1 -6235.805,E2 -6235.805} C_VEL
LIN {X 0,Y 495.831,Z 96.85,A -85,B 0,C 180,E1 -6236.522,E2 -6236.522} C_VEL
LIN {X 0,Y 495.766,Z 96.855,A -85,B 0,C 180,E1 -6239.746,E2 -6239.746} C_VEL
LIN {X 0,Y 495.767,Z 96.854,A -85,B 0,C 180,E1 -6242.594,E2 -6242.594} C_VEL
LIN {X 0,Y 495.748,Z 96.854,A -85,B 0,C 180,E1 -6245.537,E2 -6245.537} C_VEL
LIN {X 0,Y 495.764,Z 96.851,A -85,B 0,C 180,E1 -6248.768,E2 -6248.768} C_VEL
LIN {X 0,Y 495.757,Z 96.858,A -85,B 0,C 180,E1 -6251.781,E2 -6251.781} C_VEL
LIN {X 0,Y 495.749,Z 96.854,A -85,B 0,C 180,E1 -6255.139,E2 -6255.139} C_VEL
LIN {X 0,Y 495.777,Z 96.851,A -85,B 0,C 180,E1 -6258.221,E2 -6258.221} C_VEL
LIN {X 0,Y 495.749,Z 96.859,A -85,B 0,C 180,E1 -6261.408,E2 -6261.408} C_VEL
LIN {X 0,Y 495.747,Z 96.853,A -85,B 0,C 180,E1 -6264.462,E2 -6264.462} C_VEL
LIN {X 0,Y 495.767,Z 96.859,A -85,B 0,C 180,E1 -6267.406,E2 -6267.406} C_VEL
LIN {X 0,Y 495.765,Z 96.851,A -85,B 0,C 180,E1 -6270.254,E2 -6270.254} C_VEL
LIN {X 0,Y 495.822,Z 96.851,A -85,B 0,C 180,E1 -6273.251,E2 -6273.251} C_VEL
LIN {X 0,Y 495.747,Z 96.854,A -85,B 0,C 180,E1 -6275.725,E2 -6275.725} C_VEL
LIN {X 0,Y 495.741,Z 96.855,A -85,B 0,C 180,E1 -6278.371,E2 -6278.371} C_VEL
LIN {X 0,Y 495.783,Z 96.857,A -85,B 0,C 180,E1 -6280.972,E2 -6280.972} C_VEL
LIN {X 0,Y 495.776,Z 96.85,A -85,B 0,C 180,E1 -6283.53,E2 -6283.53} C_VEL
LIN {X 0,Y 495.793,Z 96.848,A -85,B 0,C 180,E1 -6286.056,E2 -6286.056} C_VEL
LIN {X 0,Y 495.85,Z 96.847,A -85,B 0,C 180,E1 -6288.555,E2 -6288.555} C_VEL
LIN {X 0,Y 495.872,Z 96.838,A -85,B 0,C 180,E1 -6291.852,E2 -6291.852} C_VEL
LIN {X 0,Y 495.89,Z 96.841,A -85,B 0,C 180,E1 -6294.307,E2 -6294.307} C_VEL
LIN {X 0,Y 495.992,Z 96.823,A -85,B 0,C 180,E1 -6297.564,E2 -6297.564} C_VEL
LIN {X 0,Y 495.982,Z 96.826,A -85,B 0,C 180,E1 -6300.812,E2 -6300.812} C_VEL
LIN {X 0,Y 495.991,Z 96.828,A -85,B 0,C 180,E1 -6302.436,E2 -6302.436} C_VEL
LIN {X 0,Y 495.881,Z 96.839,A -85,B 0,C 180,E1 -6305.694,E2 -6305.694} C_VEL
LIN {X 0,Y 495.842,Z 96.841,A -85,B 0,C 180,E1 -6308.97,E2 -6308.97} C_VEL
LIN {X 0,Y 495.828,Z 96.85,A -85,B 0,C 180,E1 -6312.035,E2 -6312.035} C_VEL
LIN {X 0,Y 495.823,Z 96.847,A -85,B 0,C 180,E1 -6315.452,E2 -6315.452} C_VEL
LIN {X 0,Y 495.776,Z 96.851,A -85,B 0,C 180,E1 -6318.237,E2 -6318.237} C_VEL
LIN {X 0,Y 495.774,Z 96.85,A -85,B 0,C 180,E1 -6320.757,E2 -6320.757} C_VEL
LIN {X 0,Y 495.742,Z 96.86,A -85,B 0,C 180,E1 -6323.388,E2 -6323.388} C_VEL
LIN {X 0,Y 495.823,Z 96.844,A -85,B 0,C 180,E1 -6326.749,E2 -6326.749} C_VEL
LIN {X 0,Y 495.765,Z 96.854,A -85,B 0,C 180,E1 -6329.747,E2 -6329.747} C_VEL
LIN {X 0,Y 495.766,Z 96.852,A -85,B 0,C 180,E1 -6332.595,E2 -6332.595} C_VEL
LIN {X 0,Y 495.747,Z 96.856,A -85,B 0,C 180,E1 -6335.538,E2 -6335.538} C_VEL
LIN {X 0,Y 495.76,Z 96.856,A -85,B 0,C 180,E1 -6338.768,E2 -6338.768} C_VEL
LIN {X 0,Y 495.756,Z 96.852,A -85,B 0,C 180,E1 -6341.781,E2 -6341.781} C_VEL
LIN {X 0,Y 495.738,Z 96.858,A -85,B 0,C 180,E1 -6345.141,E2 -6345.141} C_VEL
LIN {X 0,Y 495.751,Z 96.855,A -85,B 0,C 180,E1 -6348.219,E2 -6348.219} C_VEL
LIN {X 0,Y 495.75,Z 96.853,A -85,B 0,C 180,E1 -6351.409,E2 -6351.409} C_VEL
LIN {X 0,Y 495.746,Z 96.861,A -85,B 0,C 180,E1 -6354.462,E2 -6354.462} C_VEL
LIN {X 0,Y 495.769,Z 96.85,A -85,B 0,C 180,E1 -6357.406,E2 -6357.406} C_VEL
LIN {X 0,Y 495.765,Z 96.858,A -85,B 0,C 180,E1 -6360.254,E2 -6360.254} C_VEL
LIN {X 0,Y 495.738,Z 96.856,A -85,B 0,C 180,E1 -6360.743,E2 -6360.743} C_VEL
LIN {X 0,Y 495.064,Z 96.938,A -85,B 0,C 180,E1 -6361.422,E2 -6361.422} C_VEL
LIN {X 0,Y 492.191,Z 97.3,A -85,B 0,C 180,E1 -6362.524,E2 -6362.524} C_VEL
LIN {X 0,Y 489.78,Z 97.598,A -85,B 0,C 180,E1 -6363.412,E2 -6363.412} C_VEL
LIN {X 0,Y 488.767,Z 97.73,A -85,B 0,C 180,E1 -6364.098,E2 -6364.098} C_VEL
LIN {X 0,Y 488.696,Z 97.735,A -85,B 0,C 180,E1 -6364.331,E2 -6364.331} C_VEL
LIN {X 0,Y 488.724,Z 97.728,A -85,B 0,C 180,E1 -6367.153,E2 -6367.153} C_VEL
LIN {X 0,Y 488.727,Z 97.735,A -85,B 0,C 180,E1 -6369.811,E2 -6369.811} C_VEL
LIN {X 0,Y 488.758,Z 97.853,A -85,B 0,C 180,E1 -6372.091,E2 -6372.091} C_VEL
LIN {X 0,Y 490.658,Z 107.387,A -85,B 0,C 180,E1 -6373.91,E2 -6373.91} C_VEL
LIN {X 0,Y 490.452,Z 117.41,A -85,B 0,C 180,E1 -6375.689,E2 -6375.689} C_VEL
LIN {X 0,Y 490.333,Z 121.409,A -85,B 0,C 180,E1 -6376.391,E2 -6376.391} C_VEL
LIN {X 0,Y 493.54,Z 137.154,A -85,B 0,C 180,E1 -6376.757,E2 -6376.757} C_VEL
LIN {X 0,Y 492.522,Z 258.189,A -85,B 0,C 180,E1 -6378.555,E2 -6378.555} C_VEL
LIN {X 0,Y 492.207,Z 272.646,A -85,B 0,C 180,E1 -6378.938,E2 -6378.938} C_VEL
LIN {X 0,Y 491.89,Z 287,A -85,B 0,C 180,E1 -6379.504,E2 -6379.504} C_VEL
LIN {X 0,Y 491.409,Z 298.895,A -85,B 0,C 180,E1 -6380.118,E2 -6380.118} C_VEL
LIN {X 0,Y 490.811,Z 311.475,A -85,B 0,C 180,E1 -6380.938,E2 -6380.938} C_VEL
LIN {X 0,Y 490.324,Z 322.916,A -85,B 0,C 180,E1 -6381.863,E2 -6381.863} C_VEL
LIN {X 0,Y 489.82,Z 334.383,A -85,B 0,C 180,E1 -6382.995,E2 -6382.995} C_VEL
LIN {X 0,Y 489.267,Z 344.67,A -85,B 0,C 180,E1 -6384.229,E2 -6384.229} C_VEL
LIN {X 0,Y 488.807,Z 353.176,A -85,B 0,C 180,E1 -6385.465,E2 -6385.465} C_VEL
LIN {X 0,Y 488.49,Z 361.342,A -85,B 0,C 180,E1 -6386.907,E2 -6386.907} C_VEL
LIN {X 0,Y 488.107,Z 367.931,A -85,B 0,C 180,E1 -6388.35,E2 -6388.35} C_VEL
LIN {X 0,Y 487.955,Z 373.783,A -85,B 0,C 180,E1 -6390,E2 -6390} C_VEL
LIN {X 0,Y 487.912,Z 378.092,A -85,B 0,C 180,E1 -6391.651,E2 -6391.651} C_VEL
LIN {X 0,Y 487.961,Z 380.974,A -85,B 0,C 180,E1 -6393.303,E2 -6393.303} C_VEL
LIN {X 0,Y 487.895,Z 382.514,A -85,B 0,C 180,E1 -6394.958,E2 -6394.958} C_VEL
LIN {X 0,Y 487.949,Z 382.728,A -85,B 0,C 180,E1 -6396.617,E2 -6396.617} C_VEL
LIN {X 0,Y 487.853,Z 381.615,A -85,B 0,C 180,E1 -6398.283,E2 -6398.283} C_VEL
LIN {X 0,Y 487.912,Z 379.14,A -85,B 0,C 180,E1 -6399.954,E2 -6399.954} C_VEL
LIN {X 0,Y 488.058,Z 375.204,A -85,B 0,C 180,E1 -6401.631,E2 -6401.631} C_VEL
LIN {X 0,Y 488.194,Z 369.651,A -85,B 0,C 180,E1 -6403.317,E2 -6403.317} C_VEL
LIN {X 0,Y 488.44,Z 363.337,A -85,B 0,C 180,E1 -6404.797,E2 -6404.797} C_VEL
LIN {X 0,Y 488.803,Z 355.431,A -85,B 0,C 180,E1 -6406.282,E2 -6406.282} C_VEL
LIN {X 0,Y 489.168,Z 347.124,A -85,B 0,C 180,E1 -6407.561,E2 -6407.561} C_VEL
LIN {X 0,Y 489.7,Z 336.915,A -85,B 0,C 180,E1 -6408.857,E2 -6408.857} C_VEL
LIN {X 0,Y 490.25,Z 325.82,A -85,B 0,C 180,E1 -6410.015,E2 -6410.015} C_VEL
LIN {X 0,Y 490.739,Z 314.561,A -85,B 0,C 180,E1 -6410.979,E2 -6410.979} C_VEL
LIN {X 0,Y 491.376,Z 302.266,A -85,B 0,C 180,E1 -6411.831,E2 -6411.831} C_VEL
LIN {X 0,Y 491.865,Z 289.68,A -85,B 0,C 180,E1 -6412.527,E2 -6412.527} C_VEL
LIN {X 0,Y 492.261,Z 275.576,A -85,B 0,C 180,E1 -6413.118,E2 -6413.118} C_VEL
LIN {X 0,Y 492.6,Z 260.732,A -85,B 0,C 180,E1 -6413.546,E2 -6413.546} C_VEL
LIN {X 0,Y 492.873,Z 238.111,A -85,B 0,C 180,E1 -6413.92,E2 -6413.92} C_VEL
LIN {X 0,Y 493.639,Z 136.385,A -85,B 0,C 180,E1 -6415.433,E2 -6415.433} C_VEL
LIN {X 0,Y 490.447,Z 121.412,A -85,B 0,C 180,E1 -6415.823,E2 -6415.823} C_VEL
LIN {X 0,Y 490.885,Z 109.595,A -85,B 0,C 180,E1 -6417.94,E2 -6417.94} C_VEL
LIN {X 0,Y 489.558,Z 101.791,A -85,B 0,C 180,E1 -6419.452,E2 -6419.452} C_VEL
LIN {X 0,Y 488.675,Z 97.742,A -85,B 0,C 180,E1 -6420.274,E2 -6420.274} C_VEL
LIN {X 0,Y 488.694,Z 97.736,A -85,B 0,C 180,E1 -6423.476,E2 -6423.476} C_VEL
LIN {X 0,Y 488.646,Z 97.74,A -85,B 0,C 180,E1 -6426.348,E2 -6426.348} C_VEL
LIN {X 0,Y 488.67,Z 97.738,A -85,B 0,C 180,E1 -6429.257,E2 -6429.257} C_VEL
LIN {X 0,Y 488.648,Z 97.739,A -85,B 0,C 180,E1 -6432.53,E2 -6432.53} C_VEL
LIN {X 0,Y 488.701,Z 97.735,A -85,B 0,C 180,E1 -6435.197,E2 -6435.197} C_VEL
LIN {X 0,Y 488.662,Z 97.737,A -85,B 0,C 180,E1 -6438.579,E2 -6438.579} C_VEL
LIN {X 0,Y 488.689,Z 97.729,A -85,B 0,C 180,E1 -6440.95,E2 -6440.95} C_VEL
LIN {X 0,Y 488.666,Z 97.736,A -85,B 0,C 180,E1 -6443.867,E2 -6443.867} C_VEL
LIN {X 0,Y 488.736,Z 97.731,A -85,B 0,C 180,E1 -6446.877,E2 -6446.877} C_VEL
LIN {X 0,Y 488.719,Z 97.728,A -85,B 0,C 180,E1 -6449.78,E2 -6449.78} C_VEL
LIN {X 0,Y 488.699,Z 97.735,A -85,B 0,C 180,E1 -6453.078,E2 -6453.078} C_VEL
LIN {X 0,Y 488.669,Z 97.737,A -85,B 0,C 180,E1 -6456.253,E2 -6456.253} C_VEL
LIN {X 0,Y 488.748,Z 97.728,A -85,B 0,C 180,E1 -6459.176,E2 -6459.176} C_VEL
LIN {X 0,Y 488.749,Z 97.722,A -85,B 0,C 180,E1 -6461.632,E2 -6461.632} C_VEL
LIN {X 0,Y 488.755,Z 97.725,A -85,B 0,C 180,E1 -6464.999,E2 -6464.999} C_VEL
LIN {X 0,Y 488.806,Z 97.726,A -85,B 0,C 180,E1 -6468.387,E2 -6468.387} C_VEL
LIN {X 0,Y 488.786,Z 97.718,A -85,B 0,C 180,E1 -6471.733,E2 -6471.733} C_VEL
LIN {X 0,Y 488.838,Z 97.72,A -85,B 0,C 180,E1 -6474.224,E2 -6474.224} C_VEL
LIN {X 0,Y 488.955,Z 97.699,A -85,B 0,C 180,E1 -6477.528,E2 -6477.528} C_VEL
LIN {X 0,Y 488.914,Z 97.701,A -85,B 0,C 180,E1 -6480.823,E2 -6480.823} C_VEL
LIN {X 0,Y 488.956,Z 97.7,A -85,B 0,C 180,E1 -6482.471,E2 -6482.471} C_VEL
LIN {X 0,Y 488.831,Z 97.717,A -85,B 0,C 180,E1 -6485.776,E2 -6485.776} C_VEL
LIN {X 0,Y 488.786,Z 97.722,A -85,B 0,C 180,E1 -6488.267,E2 -6488.267} C_VEL
LIN {X 0,Y 488.806,Z 97.721,A -85,B 0,C 180,E1 -6491.612,E2 -6491.612} C_VEL
LIN {X 0,Y 488.762,Z 97.727,A -85,B 0,C 180,E1 -6495,E2 -6495} C_VEL
LIN {X 0,Y 488.756,Z 97.724,A -85,B 0,C 180,E1 -6498.442,E2 -6498.442} C_VEL
LIN {X 0,Y 488.707,Z 97.732,A -85,B 0,C 180,E1 -6501.071,E2 -6501.071} C_VEL
LIN {X 0,Y 488.689,Z 97.732,A -85,B 0,C 180,E1 -6503.746,E2 -6503.746} C_VEL
LIN {X 0,Y 488.793,Z 97.727,A -85,B 0,C 180,E1 -6506.944,E2 -6506.944} C_VEL
LIN {X 0,Y 488.711,Z 97.732,A -85,B 0,C 180,E1 -6510.363,E2 -6510.363} C_VEL
LIN {X 0,Y 488.736,Z 97.728,A -85,B 0,C 180,E1 -6513.484,E2 -6513.484} C_VEL
LIN {X 0,Y 488.683,Z 97.736,A -85,B 0,C 180,E1 -6516.355,E2 -6516.355} C_VEL
LIN {X 0,Y 488.701,Z 97.725,A -85,B 0,C 180,E1 -6519.254,E2 -6519.254} C_VEL
LIN {X 0,Y 488.708,Z 97.73,A -85,B 0,C 180,E1 -6521.6,E2 -6521.6} C_VEL
LIN {X 0,Y 488.702,Z 97.731,A -85,B 0,C 180,E1 -6524.803,E2 -6524.803} C_VEL
LIN {X 0,Y 488.693,Z 97.733,A -85,B 0,C 180,E1 -6527.474,E2 -6527.474} C_VEL
LIN {X 0,Y 488.734,Z 97.73,A -85,B 0,C 180,E1 -6529.677,E2 -6529.677} C_VEL
LIN {X 0,Y 488.68,Z 97.733,A -85,B 0,C 180,E1 -6532.841,E2 -6532.841} C_VEL
LIN {X 0,Y 488.732,Z 97.732,A -85,B 0,C 180,E1 -6535.887,E2 -6535.887} C_VEL
LIN {X 0,Y 488.693,Z 97.733,A -85,B 0,C 180,E1 -6538.82,E2 -6538.82} C_VEL
LIN {X 0,Y 488.746,Z 97.733,A -85,B 0,C 180,E1 -6541.671,E2 -6541.671} C_VEL
LIN {X 0,Y 488.779,Z 97.759,A -85,B 0,C 180,E1 -6543.009,E2 -6543.009} C_VEL
LIN {X 0,Y 491.505,Z 110.54,A -85,B 0,C 180,E1 -6545.276,E2 -6545.276} C_VEL
LIN {X 0,Y 491.237,Z 120.231,A -85,B 0,C 180,E1 -6546.831,E2 -6546.831} C_VEL
LIN {X 0,Y 490.366,Z 139.632,A -85,B 0,C 180,E1 -6549.881,E2 -6549.881} C_VEL
LIN {X 0,Y 490.327,Z 141.819,A -85,B 0,C 180,E1 -6550.224,E2 -6550.224} C_VEL
LIN {X 0,Y 493.511,Z 159.594,A -85,B 0,C 180,E1 -6550.64,E2 -6550.64} C_VEL
LIN {X 0,Y 492.589,Z 279.122,A -85,B 0,C 180,E1 -6552.431,E2 -6552.431} C_VEL
LIN {X 0,Y 492.22,Z 293.22,A -85,B 0,C 180,E1 -6552.793,E2 -6552.793} C_VEL
LIN {X 0,Y 491.743,Z 307.455,A -85,B 0,C 180,E1 -6553.337,E2 -6553.337} C_VEL
LIN {X 0,Y 491.253,Z 320.608,A -85,B 0,C 180,E1 -6554.014,E2 -6554.014} C_VEL
LIN {X 0,Y 490.636,Z 333.322,A -85,B 0,C 180,E1 -6554.846,E2 -6554.846} C_VEL
LIN {X 0,Y 490.06,Z 344.908,A -85,B 0,C 180,E1 -6555.783,E2 -6555.783} C_VEL
LIN {X 0,Y 489.514,Z 356.519,A -85,B 0,C 180,E1 -6556.931,E2 -6556.931} C_VEL
LIN {X 0,Y 489.075,Z 366.027,A -85,B 0,C 180,E1 -6558.069,E2 -6558.069} C_VEL
LIN {X 0,Y 488.675,Z 375.499,A -85,B 0,C 180,E1 -6559.434,E2 -6559.434} C_VEL
LIN {X 0,Y 488.325,Z 383.727,A -85,B 0,C 180,E1 -6560.891,E2 -6560.891} C_VEL
LIN {X 0,Y 488.144,Z 389.495,A -85,B 0,C 180,E1 -6562.139,E2 -6562.139} C_VEL
LIN {X 0,Y 488.002,Z 394.864,A -85,B 0,C 180,E1 -6563.57,E2 -6563.57} C_VEL
LIN {X 0,Y 487.957,Z 399.125,A -85,B 0,C 180,E1 -6565.042,E2 -6565.042} C_VEL
LIN {X 0,Y 487.955,Z 402.536,A -85,B 0,C 180,E1 -6566.697,E2 -6566.697} C_VEL
LIN {X 0,Y 487.888,Z 404.553,A -85,B 0,C 180,E1 -6568.349,E2 -6568.349} C_VEL
LIN {X 0,Y 487.819,Z 405.222,A -85,B 0,C 180,E1 -6570,E2 -6570} C_VEL
LIN {X 0,Y 487.888,Z 404.556,A -85,B 0,C 180,E1 -6571.651,E2 -6571.651} C_VEL
LIN {X 0,Y 487.954,Z 402.54,A -85,B 0,C 180,E1 -6573.303,E2 -6573.303} C_VEL
LIN {X 0,Y 487.957,Z 399.124,A -85,B 0,C 180,E1 -6574.957,E2 -6574.957} C_VEL
LIN {X 0,Y 488.033,Z 394.206,A -85,B 0,C 180,E1 -6576.615,E2 -6576.615} C_VEL
LIN {X 0,Y 488.223,Z 387.643,A -85,B 0,C 180,E1 -6578.276,E2 -6578.276} C_VEL
LIN {X 0,Y 488.451,Z 380.333,A -85,B 0,C 180,E1 -6579.733,E2 -6579.733} C_VEL
LIN {X 0,Y 488.87,Z 371.272,A -85,B 0,C 180,E1 -6581.191,E2 -6581.191} C_VEL
LIN {X 0,Y 489.235,Z 361.759,A -85,B 0,C 180,E1 -6582.443,E2 -6582.443} C_VEL
LIN {X 0,Y 489.74,Z 351.219,A -85,B 0,C 180,E1 -6583.591,E2 -6583.591} C_VEL
LIN {X 0,Y 490.266,Z 339.578,A -85,B 0,C 180,E1 -6584.635,E2 -6584.635} C_VEL
LIN {X 0,Y 490.869,Z 326.652,A -85,B 0,C 180,E1 -6585.572,E2 -6585.572} C_VEL
LIN {X 0,Y 491.499,Z 312.993,A -85,B 0,C 180,E1 -6586.35,E2 -6586.35} C_VEL
LIN {X 0,Y 491.872,Z 299.44,A -85,B 0,C 180,E1 -6586.941,E2 -6586.941} C_VEL
LIN {X 0,Y 492.333,Z 284.767,A -85,B 0,C 180,E1 -6587.385,E2 -6587.385} C_VEL
LIN {X 0,Y 492.572,Z 268.932,A -85,B 0,C 180,E1 -6587.676,E2 -6587.676} C_VEL
LIN {X 0,Y 493.294,Z 159.505,A -85,B 0,C 180,E1 -6589.288,E2 -6589.288} C_VEL
LIN {X 0,Y 490.224,Z 141.874,A -85,B 0,C 180,E1 -6589.677,E2 -6589.677} C_VEL
LIN {X 0,Y 490.923,Z 122.088,A -85,B 0,C 180,E1 -6592.739,E2 -6592.739} C_VEL
LIN {X 0,Y 491.395,Z 110.79,A -85,B 0,C 180,E1 -6594.504,E2 -6594.504} C_VEL
LIN {X 0,Y 488.921,Z 98.406,A -85,B 0,C 180,E1 -6596.614,E2 -6596.614} C_VEL
LIN {X 0,Y 488.785,Z 97.728,A -85,B 0,C 180,E1 -6596.774,E2 -6596.774} C_VEL
LIN {X 0,Y 488.724,Z 97.731,A -85,B 0,C 180,E1 -6599.27,E2 -6599.27} C_VEL
LIN {X 0,Y 488.703,Z 97.739,A -85,B 0,C 180,E1 -6602.147,E2 -6602.147} C_VEL
LIN {X 0,Y 488.717,Z 97.729,A -85,B 0,C 180,E1 -6605.115,E2 -6605.115} C_VEL
LIN {X 0,Y 488.68,Z 97.739,A -85,B 0,C 180,E1 -6608.2,E2 -6608.2} C_VEL
LIN {X 0,Y 488.717,Z 97.732,A -85,B 0,C 180,E1 -6610.344,E2 -6610.344} C_VEL
LIN {X 0,Y 488.686,Z 97.738,A -85,B 0,C 180,E1 -6613.654,E2 -6613.654} C_VEL
LIN {X 0,Y 488.716,Z 97.73,A -85,B 0,C 180,E1 -6616.349,E2 -6616.349} C_VEL
LIN {X 0,Y 488.718,Z 97.729,A -85,B 0,C 180,E1 -6618.585,E2 -6618.585} C_VEL
LIN {X 0,Y 488.678,Z 97.739,A -85,B 0,C 180,E1 -6621.8,E2 -6621.8} C_VEL
LIN {X 0,Y 488.722,Z 97.731,A -85,B 0,C 180,E1 -6625.052,E2 -6625.052} C_VEL
LIN {X 0,Y 488.703,Z 97.731,A -85,B 0,C 180,E1 -6628.046,E2 -6628.046} C_VEL
LIN {X 0,Y 488.722,Z 97.73,A -85,B 0,C 180,E1 -6630.73,E2 -6630.73} C_VEL
LIN {X 0,Y 488.756,Z 97.728,A -85,B 0,C 180,E1 -6633.528,E2 -6633.528} C_VEL
LIN {X 0,Y 488.688,Z 97.733,A -85,B 0,C 180,E1 -6636.254,E2 -6636.254} C_VEL
LIN {X 0,Y 488.745,Z 97.731,A -85,B 0,C 180,E1 -6639.176,E2 -6639.176} C_VEL
LIN {X 0,Y 488.758,Z 97.724,A -85,B 0,C 180,E1 -6641.628,E2 -6641.628} C_VEL
LIN {X 0,Y 488.761,Z 97.729,A -85,B 0,C 180,E1 -6645,E2 -6645} C_VEL
LIN {X 0,Y 488.804,Z 97.722,A -85,B 0,C 180,E1 -6648.388,E2 -6648.388} C_VEL
LIN {X 0,Y 488.816,Z 97.717,A -85,B 0,C 180,E1 -6651.734,E2 -6651.734} C_VEL
LIN {X 0,Y 488.848,Z 97.717,A -85,B 0,C 180,E1 -6654.224,E2 -6654.224} C_VEL
LIN {X 0,Y 488.96,Z 97.699,A -85,B 0,C 180,E1 -6657.529,E2 -6657.529} C_VEL
LIN {X 0,Y 488.934,Z 97.703,A -85,B 0,C 180,E1 -6660.824,E2 -6660.824} C_VEL
LIN {X 0,Y 488.959,Z 97.703,A -85,B 0,C 180,E1 -6662.472,E2 -6662.472} C_VEL
LIN {X 0,Y 488.838,Z 97.717,A -85,B 0,C 180,E1 -6665.776,E2 -6665.776} C_VEL
LIN {X 0,Y 488.817,Z 97.721,A -85,B 0,C 180,E1 -6668.267,E2 -6668.267} C_VEL
LIN {X 0,Y 488.805,Z 97.722,A -85,B 0,C 180,E1 -6671.613,E2 -6671.613} C_VEL
LIN {X 0,Y 488.761,Z 97.723,A -85,B 0,C 180,E1 -6675.001,E2 -6675.001} C_VEL
LIN {X 0,Y 488.745,Z 97.726,A -85,B 0,C 180,E1 -6678.443,E2 -6678.443} C_VEL
LIN {X 0,Y 488.706,Z 97.732,A -85,B 0,C 180,E1 -6681.071,E2 -6681.071} C_VEL
LIN {X 0,Y 488.679,Z 97.739,A -85,B 0,C 180,E1 -6683.746,E2 -6683.746} C_VEL
LIN {X 0,Y 488.791,Z 97.722,A -85,B 0,C 180,E1 -6686.944,E2 -6686.944} C_VEL
LIN {X 0,Y 488.708,Z 97.73,A -85,B 0,C 180,E1 -6690.363,E2 -6690.363} C_VEL
LIN {X 0,Y 488.729,Z 97.732,A -85,B 0,C 180,E1 -6693.483,E2 -6693.483} C_VEL
LIN {X 0,Y 488.682,Z 97.734,A -85,B 0,C 180,E1 -6696.355,E2 -6696.355} C_VEL
LIN {X 0,Y 488.698,Z 97.736,A -85,B 0,C 180,E1 -6699.255,E2 -6699.255} C_VEL
LIN {X 0,Y 488.707,Z 97.731,A -85,B 0,C 180,E1 -6701.6,E2 -6701.6} C_VEL
LIN {X 0,Y 488.702,Z 97.739,A -85,B 0,C 180,E1 -6704.803,E2 -6704.803} C_VEL
LIN {X 0,Y 488.689,Z 97.733,A -85,B 0,C 180,E1 -6707.474,E2 -6707.474} C_VEL
LIN {X 0,Y 488.702,Z 97.737,A -85,B 0,C 180,E1 -6710.746,E2 -6710.746} C_VEL
LIN {X 0,Y 488.671,Z 97.735,A -85,B 0,C 180,E1 -6713.868,E2 -6713.868} C_VEL
LIN {X 0,Y 488.74,Z 97.728,A -85,B 0,C 180,E1 -6716.878,E2 -6716.878} C_VEL
LIN {X 0,Y 488.726,Z 97.729,A -85,B 0,C 180,E1 -6719.781,E2 -6719.781} C_VEL
LIN {X 0,Y 488.716,Z 97.729,A -85,B 0,C 180,E1 -6723.075,E2 -6723.075} C_VEL
LIN {X 0,Y 488.696,Z 97.735,A -85,B 0,C 180,E1 -6724.331,E2 -6724.331} C_VEL
LIN {X 0,Y 488.06,Z 97.819,A -85,B 0,C 180,E1 -6725.019,E2 -6725.019} C_VEL
LIN {X 0,Y 485.212,Z 98.175,A -85,B 0,C 180,E1 -6726.136,E2 -6726.136} C_VEL
LIN {X 0,Y 482.779,Z 98.474,A -85,B 0,C 180,E1 -6727.036,E2 -6727.036} C_VEL
LIN {X 0,Y 481.727,Z 98.603,A -85,B 0,C 180,E1 -6727.731,E2 -6727.731} C_VEL
LIN {X 0,Y 481.638,Z 98.613,A -85,B 0,C 180,E1 -6727.967,E2 -6727.967} C_VEL
LIN {X 0,Y 481.705,Z 98.609,A -85,B 0,C 180,E1 -6730.393,E2 -6730.393} C_VEL
LIN {X 0,Y 481.717,Z 98.724,A -85,B 0,C 180,E1 -6731.881,E2 -6731.881} C_VEL
LIN {X 0,Y 483.789,Z 109.594,A -85,B 0,C 180,E1 -6733.978,E2 -6733.978} C_VEL
LIN {X 0,Y 483.424,Z 121.574,A -85,B 0,C 180,E1 -6736.121,E2 -6736.121} C_VEL
LIN {X 0,Y 486.779,Z 137.913,A -85,B 0,C 180,E1 -6736.507,E2 -6736.507} C_VEL
LIN {X 0,Y 485.732,Z 258.055,A -85,B 0,C 180,E1 -6738.313,E2 -6738.313} C_VEL
LIN {X 0,Y 485.409,Z 272.626,A -85,B 0,C 180,E1 -6738.702,E2 -6738.702} C_VEL
LIN {X 0,Y 485.072,Z 286.482,A -85,B 0,C 180,E1 -6739.249,E2 -6739.249} C_VEL
LIN {X 0,Y 484.554,Z 298.532,A -85,B 0,C 180,E1 -6739.871,E2 -6739.871} C_VEL
LIN {X 0,Y 483.95,Z 311.215,A -85,B 0,C 180,E1 -6740.703,E2 -6740.703} C_VEL
LIN {X 0,Y 483.367,Z 323.897,A -85,B 0,C 180,E1 -6741.745,E2 -6741.745} C_VEL
LIN {X 0,Y 482.845,Z 335.232,A -85,B 0,C 180,E1 -6742.893,E2 -6742.893} C_VEL
LIN {X 0,Y 482.255,Z 345.402,A -85,B 0,C 180,E1 -6744.145,E2 -6744.145} C_VEL
LIN {X 0,Y 481.774,Z 353.82,A -85,B 0,C 180,E1 -6745.398,E2 -6745.398} C_VEL
LIN {X 0,Y 481.41,Z 361.878,A -85,B 0,C 180,E1 -6746.862,E2 -6746.862} C_VEL
LIN {X 0,Y 481.029,Z 368.39,A -85,B 0,C 180,E1 -6748.326,E2 -6748.326} C_VEL
LIN {X 0,Y 481.035,Z 372.886,A -85,B 0,C 180,E1 -6749.582,E2 -6749.582} C_VEL
LIN {X 0,Y 480.837,Z 376.482,A -85,B 0,C 180,E1 -6750.838,E2 -6750.838} C_VEL
LIN {X 0,Y 480.847,Z 380.003,A -85,B 0,C 180,E1 -6752.513,E2 -6752.513} C_VEL
LIN {X 0,Y 480.882,Z 381.242,A -85,B 0,C 180,E1 -6753.352,E2 -6753.352} C_VEL
LIN {X 0,Y 480.819,Z 382.721,A -85,B 0,C 180,E1 -6755.031,E2 -6755.031} C_VEL
LIN {X 0,Y 480.867,Z 382.875,A -85,B 0,C 180,E1 -6756.715,E2 -6756.715} C_VEL
LIN {X 0,Y 480.767,Z 381.702,A -85,B 0,C 180,E1 -6758.406,E2 -6758.406} C_VEL
LIN {X 0,Y 480.827,Z 379.157,A -85,B 0,C 180,E1 -6760.102,E2 -6760.102} C_VEL
LIN {X 0,Y 481.007,Z 375.134,A -85,B 0,C 180,E1 -6761.804,E2 -6761.804} C_VEL
LIN {X 0,Y 481.155,Z 369.512,A -85,B 0,C 180,E1 -6763.515,E2 -6763.515} C_VEL
LIN {X 0,Y 481.404,Z 363.127,A -85,B 0,C 180,E1 -6765.019,E2 -6765.019} C_VEL
LIN {X 0,Y 481.813,Z 355.142,A -85,B 0,C 180,E1 -6766.525,E2 -6766.525} C_VEL
LIN {X 0,Y 482.241,Z 346.746,A -85,B 0,C 180,E1 -6767.821,E2 -6767.821} C_VEL
LIN {X 0,Y 482.784,Z 336.944,A -85,B 0,C 180,E1 -6769.076,E2 -6769.076} C_VEL
LIN {X 0,Y 483.345,Z 326.308,A -85,B 0,C 180,E1 -6770.202,E2 -6770.202} C_VEL
LIN {X 0,Y 483.887,Z 315.132,A -85,B 0,C 180,E1 -6771.179,E2 -6771.179} C_VEL
LIN {X 0,Y 484.563,Z 302.429,A -85,B 0,C 180,E1 -6772.076,E2 -6772.076} C_VEL
LIN {X 0,Y 485.118,Z 289.411,A -85,B 0,C 180,E1 -6772.801,E2 -6772.801} C_VEL
LIN {X 0,Y 485.547,Z 275.169,A -85,B 0,C 180,E1 -6773.4,E2 -6773.4} C_VEL
LIN {X 0,Y 485.882,Z 261.217,A -85,B 0,C 180,E1 -6773.806,E2 -6773.806} C_VEL
LIN {X 0,Y 486.177,Z 239.263,A -85,B 0,C 180,E1 -6774.178,E2 -6774.178} C_VEL
LIN {X 0,Y 487.053,Z 137.6,A -85,B 0,C 180,E1 -6775.709,E2 -6775.709} C_VEL
LIN {X 0,Y 483.612,Z 121.562,A -85,B 0,C 180,E1 -6776.138,E2 -6776.138} C_VEL
LIN {X 0,Y 483.965,Z 110.463,A -85,B 0,C 180,E1 -6778.161,E2 -6778.161} C_VEL
LIN {X 0,Y 481.967,Z 100.201,A -85,B 0,C 180,E1 -6780.204,E2 -6780.204} C_VEL
LIN {X 0,Y 481.612,Z 98.621,A -85,B 0,C 180,E1 -6780.574,E2 -6780.574} C_VEL
LIN {X 0,Y 481.65,Z 98.616,A -85,B 0,C 180,E1 -6783.724,E2 -6783.724} C_VEL
LIN {X 0,Y 481.605,Z 98.615,A -85,B 0,C 180,E1 -6786.749,E2 -6786.749} C_VEL
LIN {X 0,Y 481.629,Z 98.619,A -85,B 0,C 180,E1 -6789.945,E2 -6789.945} C_VEL
LIN {X 0,Y 481.615,Z 98.619,A -85,B 0,C 180,E1 -6793.303,E2 -6793.303} C_VEL
LIN {X 0,Y 481.653,Z 98.61,A -85,B 0,C 180,E1 -6795.642,E2 -6795.642} C_VEL
LIN {X 0,Y 481.624,Z 98.616,A -85,B 0,C 180,E1 -6798.954,E2 -6798.954} C_VEL
LIN {X 0,Y 481.635,Z 98.613,A -85,B 0,C 180,E1 -6801.996,E2 -6801.996} C_VEL
LIN {X 0,Y 481.683,Z 98.612,A -85,B 0,C 180,E1 -6805.317,E2 -6805.317} C_VEL
LIN {X 0,Y 481.644,Z 98.611,A -85,B 0,C 180,E1 -6808.311,E2 -6808.311} C_VEL
LIN {X 0,Y 481.661,Z 98.614,A -85,B 0,C 180,E1 -6811.216,E2 -6811.216} C_VEL
LIN {X 0,Y 481.63,Z 98.609,A -85,B 0,C 180,E1 -6814.038,E2 -6814.038} C_VEL
LIN {X 0,Y 481.654,Z 98.613,A -85,B 0,C 180,E1 -6816.818,E2 -6816.818} C_VEL
LIN {X 0,Y 481.696,Z 98.605,A -85,B 0,C 180,E1 -6819.502,E2 -6819.502} C_VEL
LIN {X 0,Y 481.689,Z 98.604,A -85,B 0,C 180,E1 -6822.158,E2 -6822.158} C_VEL
LIN {X 0,Y 481.739,Z 98.601,A -85,B 0,C 180,E1 -6824.775,E2 -6824.775} C_VEL
LIN {X 0,Y 481.752,Z 98.601,A -85,B 0,C 180,E1 -6828.215,E2 -6828.215} C_VEL
LIN {X 0,Y 481.74,Z 98.594,A -85,B 0,C 180,E1 -6831.611,E2 -6831.611} C_VEL
LIN {X 0,Y 481.797,Z 98.598,A -85,B 0,C 180,E1 -6834.139,E2 -6834.139} C_VEL
LIN {X 0,Y 481.921,Z 98.575,A -85,B 0,C 180,E1 -6837.492,E2 -6837.492} C_VEL
LIN {X 0,Y 481.941,Z 98.577,A -85,B 0,C 180,E1 -6840,E2 -6840} C_VEL
LIN {X 0,Y 481.922,Z 98.576,A -85,B 0,C 180,E1 -6842.507,E2 -6842.507} C_VEL
LIN {X 0,Y 481.79,Z 98.593,A -85,B 0,C 180,E1 -6845.861,E2 -6845.861} C_VEL
LIN {X 0,Y 481.741,Z 98.599,A -85,B 0,C 180,E1 -6848.389,E2 -6848.389} C_VEL
LIN {X 0,Y 481.751,Z 98.6,A -85,B 0,C 180,E1 -6851.785,E2 -6851.785} C_VEL
LIN {X 0,Y 481.743,Z 98.603,A -85,B 0,C 180,E1 -6855.224,E2 -6855.224} C_VEL
LIN {X 0,Y 481.713,Z 98.603,A -85,B 0,C 180,E1 -6858.722,E2 -6858.722} C_VEL
LIN {X 0,Y 481.647,Z 98.614,A -85,B 0,C 180,E1 -6861.395,E2 -6861.395} C_VEL
LIN {X 0,Y 481.674,Z 98.605,A -85,B 0,C 180,E1 -6864.113,E2 -6864.113} C_VEL
LIN {X 0,Y 481.747,Z 98.602,A -85,B 0,C 180,E1 -6867.139,E2 -6867.139} C_VEL
LIN {X 0,Y 481.68,Z 98.605,A -85,B 0,C 180,E1 -6869.741,E2 -6869.741} C_VEL
LIN {X 0,Y 481.673,Z 98.611,A -85,B 0,C 180,E1 -6872.674,E2 -6872.674} C_VEL
LIN {X 0,Y 481.638,Z 98.609,A -85,B 0,C 180,E1 -6875.709,E2 -6875.709} C_VEL
LIN {X 0,Y 481.671,Z 98.603,A -85,B 0,C 180,E1 -6878.859,E2 -6878.859} C_VEL
LIN {X 0,Y 481.654,Z 98.611,A -85,B 0,C 180,E1 -6881.913,E2 -6881.913} C_VEL
LIN {X 0,Y 481.655,Z 98.608,A -85,B 0,C 180,E1 -6884.458,E2 -6884.458} C_VEL
LIN {X 0,Y 481.648,Z 98.614,A -85,B 0,C 180,E1 -6887.839,E2 -6887.839} C_VEL
LIN {X 0,Y 481.682,Z 98.606,A -85,B 0,C 180,E1 -6890.651,E2 -6890.651} C_VEL
LIN {X 0,Y 481.628,Z 98.613,A -85,B 0,C 180,E1 -6893.376,E2 -6893.376} C_VEL
LIN {X 0,Y 481.711,Z 98.601,A -85,B 0,C 180,E1 -6896.33,E2 -6896.33} C_VEL
LIN {X 0,Y 481.652,Z 98.613,A -85,B 0,C 180,E1 -6899.417,E2 -6899.417} C_VEL
LIN {X 0,Y 481.71,Z 98.607,A -85,B 0,C 180,E1 -6902.559,E2 -6902.559} C_VEL
LIN {X 0,Y 481.77,Z 98.815,A -85,B 0,C 180,E1 -6902.757,E2 -6902.757} C_VEL
LIN {X 0,Y 484.602,Z 111.936,A -85,B 0,C 180,E1 -6905.129,E2 -6905.129} C_VEL
LIN {X 0,Y 484.587,Z 117.463,A -85,B 0,C 180,E1 -6906.041,E2 -6906.041} C_VEL
LIN {X 0,Y 483.633,Z 136.834,A -85,B 0,C 180,E1 -6909.144,E2 -6909.144} C_VEL
LIN {X 0,Y 483.41,Z 141.644,A -85,B 0,C 180,E1 -6909.906,E2 -6909.906} C_VEL
LIN {X 0,Y 486.904,Z 160.847,A -85,B 0,C 180,E1 -6910.369,E2 -6910.369} C_VEL
LIN {X 0,Y 485.844,Z 279.773,A -85,B 0,C 180,E1 -6912.179,E2 -6912.179} C_VEL
LIN {X 0,Y 485.432,Z 294.221,A -85,B 0,C 180,E1 -6912.569,E2 -6912.569} C_VEL
LIN {X 0,Y 484.943,Z 307.767,A -85,B 0,C 180,E1 -6913.103,E2 -6913.103} C_VEL
LIN {X 0,Y 484.42,Z 320.862,A -85,B 0,C 180,E1 -6913.792,E2 -6913.792} C_VEL
LIN {X 0,Y 483.778,Z 333.371,A -85,B 0,C 180,E1 -6914.626,E2 -6914.626} C_VEL
LIN {X 0,Y 483.131,Z 344.911,A -85,B 0,C 180,E1 -6915.575,E2 -6915.575} C_VEL
LIN {X 0,Y 482.56,Z 356.484,A -85,B 0,C 180,E1 -6916.739,E2 -6916.739} C_VEL
LIN {X 0,Y 482.048,Z 366.617,A -85,B 0,C 180,E1 -6917.978,E2 -6917.978} C_VEL
LIN {X 0,Y 481.658,Z 375.414,A -85,B 0,C 180,E1 -6919.278,E2 -6919.278} C_VEL
LIN {X 0,Y 481.283,Z 383.617,A -85,B 0,C 180,E1 -6920.756,E2 -6920.756} C_VEL
LIN {X 0,Y 481.075,Z 389.376,A -85,B 0,C 180,E1 -6922.022,E2 -6922.022} C_VEL
LIN {X 0,Y 480.916,Z 395.103,A -85,B 0,C 180,E1 -6923.584,E2 -6923.584} C_VEL
LIN {X 0,Y 480.886,Z 398.983,A -85,B 0,C 180,E1 -6924.969,E2 -6924.969} C_VEL
LIN {X 0,Y 480.86,Z 402.386,A -85,B 0,C 180,E1 -6926.648,E2 -6926.648} C_VEL
LIN {X 0,Y 480.789,Z 404.397,A -85,B 0,C 180,E1 -6928.325,E2 -6928.325} C_VEL
LIN {X 0,Y 480.743,Z 405.059,A -85,B 0,C 180,E1 -6930,E2 -6930} C_VEL
LIN {X 0,Y 480.789,Z 404.385,A -85,B 0,C 180,E1 -6931.675,E2 -6931.675} C_VEL
LIN {X 0,Y 480.86,Z 402.363,A -85,B 0,C 180,E1 -6933.351,E2 -6933.351} C_VEL
LIN {X 0,Y 480.887,Z 398.94,A -85,B 0,C 180,E1 -6935.03,E2 -6935.03} C_VEL
LIN {X 0,Y 480.957,Z 394.012,A -85,B 0,C 180,E1 -6936.713,E2 -6936.713} C_VEL
LIN {X 0,Y 481.142,Z 387.434,A -85,B 0,C 180,E1 -6938.399,E2 -6938.399} C_VEL
LIN {X 0,Y 481.383,Z 380.108,A -85,B 0,C 180,E1 -6939.878,E2 -6939.878} C_VEL
LIN {X 0,Y 481.856,Z 371.023,A -85,B 0,C 180,E1 -6941.356,E2 -6941.356} C_VEL
LIN {X 0,Y 482.257,Z 361.483,A -85,B 0,C 180,E1 -6942.626,E2 -6942.626} C_VEL
LIN {X 0,Y 482.804,Z 350.914,A -85,B 0,C 180,E1 -6943.79,E2 -6943.79} C_VEL
LIN {X 0,Y 483.361,Z 339.236,A -85,B 0,C 180,E1 -6944.848,E2 -6944.848} C_VEL
LIN {X 0,Y 483.988,Z 326.26,A -85,B 0,C 180,E1 -6945.799,E2 -6945.799} C_VEL
LIN {X 0,Y 484.558,Z 314.199,A -85,B 0,C 180,E1 -6946.501,E2 -6946.501} C_VEL
LIN {X 0,Y 485.021,Z 300.065,A -85,B 0,C 180,E1 -6947.139,E2 -6947.139} C_VEL
LIN {X 0,Y 485.479,Z 286.318,A -85,B 0,C 180,E1 -6947.578,E2 -6947.578} C_VEL
LIN {X 0,Y 485.728,Z 271.227,A -85,B 0,C 180,E1 -6947.879,E2 -6947.879} C_VEL
LIN {X 0,Y 486.533,Z 160.187,A -85,B 0,C 180,E1 -6949.535,E2 -6949.535} C_VEL
LIN {X 0,Y 483.278,Z 141.647,A -85,B 0,C 180,E1 -6949.962,E2 -6949.962} C_VEL
LIN {X 0,Y 484.232,Z 119.127,A -85,B 0,C 180,E1 -6953.498,E2 -6953.498} C_VEL
LIN {X 0,Y 484.453,Z 111.901,A -85,B 0,C 180,E1 -6954.65,E2 -6954.65} C_VEL
LIN {X 0,Y 481.749,Z 98.602,A -85,B 0,C 180,E1 -6956.97,E2 -6956.97} C_VEL
LIN {X 0,Y 481.679,Z 98.611,A -85,B 0,C 180,E1 -6959.741,E2 -6959.741} C_VEL
LIN {X 0,Y 481.672,Z 98.609,A -85,B 0,C 180,E1 -6962.674,E2 -6962.674} C_VEL
LIN {X 0,Y 481.636,Z 98.614,A -85,B 0,C 180,E1 -6965.709,E2 -6965.709} C_VEL
LIN {X 0,Y 481.671,Z 98.607,A -85,B 0,C 180,E1 -6968.859,E2 -6968.859} C_VEL
LIN {X 0,Y 481.653,Z 98.617,A -85,B 0,C 180,E1 -6971.913,E2 -6971.913} C_VEL
LIN {X 0,Y 481.659,Z 98.609,A -85,B 0,C 180,E1 -6974.457,E2 -6974.457} C_VEL
LIN {X 0,Y 481.689,Z 98.604,A -85,B 0,C 180,E1 -6976.846,E2 -6976.846} C_VEL
LIN {X 0,Y 481.676,Z 98.609,A -85,B 0,C 180,E1 -6980.06,E2 -6980.06} C_VEL
LIN {X 0,Y 481.624,Z 98.617,A -85,B 0,C 180,E1 -6983.253,E2 -6983.253} C_VEL
LIN {X 0,Y 481.708,Z 98.602,A -85,B 0,C 180,E1 -6986.33,E2 -6986.33} C_VEL
LIN {X 0,Y 481.65,Z 98.616,A -85,B 0,C 180,E1 -6989.417,E2 -6989.417} C_VEL
LIN {X 0,Y 481.699,Z 98.603,A -85,B 0,C 180,E1 -6992.168,E2 -6992.168} C_VEL
LIN {X 0,Y 481.716,Z 98.607,A -85,B 0,C 180,E1 -6994.97,E2 -6994.97} C_VEL
LIN {X 0,Y 481.648,Z 98.61,A -85,B 0,C 180,E1 -6997.705,E2 -6997.705} C_VEL
LIN {X 0,Y 481.704,Z 98.604,A -85,B 0,C 180,E1 -7000.393,E2 -7000.393} C_VEL
LIN {X 0,Y 481.687,Z 98.61,A -85,B 0,C 180,E1 -7003.034,E2 -7003.034} C_VEL
LIN {X 0,Y 481.689,Z 98.604,A -85,B 0,C 180,E1 -7005.639,E2 -7005.639} C_VEL
LIN {X 0,Y 481.75,Z 98.599,A -85,B 0,C 180,E1 -7008.215,E2 -7008.215} C_VEL
LIN {X 0,Y 481.762,Z 98.595,A -85,B 0,C 180,E1 -7011.612,E2 -7011.612} C_VEL
LIN {X 0,Y 481.809,Z 98.593,A -85,B 0,C 180,E1 -7014.14,E2 -7014.14} C_VEL
LIN {X 0,Y 481.927,Z 98.575,A -85,B 0,C 180,E1 -7017.493,E2 -7017.493} C_VEL
LIN {X 0,Y 481.885,Z 98.581,A -85,B 0,C 180,E1 -7020.836,E2 -7020.836} C_VEL
LIN {X 0,Y 481.926,Z 98.579,A -85,B 0,C 180,E1 -7022.508,E2 -7022.508} C_VEL
LIN {X 0,Y 481.797,Z 98.596,A -85,B 0,C 180,E1 -7025.861,E2 -7025.861} C_VEL
LIN {X 0,Y 481.762,Z 98.599,A -85,B 0,C 180,E1 -7028.388,E2 -7028.388} C_VEL
LIN {X 0,Y 481.75,Z 98.603,A -85,B 0,C 180,E1 -7031.785,E2 -7031.785} C_VEL
LIN {X 0,Y 481.742,Z 98.599,A -85,B 0,C 180,E1 -7035.224,E2 -7035.224} C_VEL
LIN {X 0,Y 481.707,Z 98.602,A -85,B 0,C 180,E1 -7038.722,E2 -7038.722} C_VEL
LIN {X 0,Y 481.646,Z 98.615,A -85,B 0,C 180,E1 -7041.395,E2 -7041.395} C_VEL
LIN {X 0,Y 481.66,Z 98.609,A -85,B 0,C 180,E1 -7044.114,E2 -7044.114} C_VEL
LIN {X 0,Y 481.746,Z 98.602,A -85,B 0,C 180,E1 -7047.139,E2 -7047.139} C_VEL
LIN {X 0,Y 481.677,Z 98.609,A -85,B 0,C 180,E1 -7049.741,E2 -7049.741} C_VEL
LIN {X 0,Y 481.67,Z 98.608,A -85,B 0,C 180,E1 -7052.675,E2 -7052.675} C_VEL
LIN {X 0,Y 481.636,Z 98.612,A -85,B 0,C 180,E1 -7055.71,E2 -7055.71} C_VEL
LIN {X 0,Y 481.668,Z 98.613,A -85,B 0,C 180,E1 -7058.86,E2 -7058.86} C_VEL
LIN {X 0,Y 481.653,Z 98.609,A -85,B 0,C 180,E1 -7061.913,E2 -7061.913} C_VEL
LIN {X 0,Y 481.655,Z 98.612,A -85,B 0,C 180,E1 -7064.458,E2 -7064.458} C_VEL
LIN {X 0,Y 481.644,Z 98.61,A -85,B 0,C 180,E1 -7067.839,E2 -7067.839} C_VEL
LIN {X 0,Y 481.661,Z 98.616,A -85,B 0,C 180,E1 -7070.655,E2 -7070.655} C_VEL
LIN {X 0,Y 481.623,Z 98.613,A -85,B 0,C 180,E1 -7073.378,E2 -7073.378} C_VEL
LIN {X 0,Y 481.712,Z 98.608,A -85,B 0,C 180,E1 -7076.33,E2 -7076.33} C_VEL
LIN {X 0,Y 481.652,Z 98.609,A -85,B 0,C 180,E1 -7079.418,E2 -7079.418} C_VEL
LIN {X 0,Y 481.667,Z 98.614,A -85,B 0,C 180,E1 -7082.166,E2 -7082.166} C_VEL
LIN {X 0,Y 481.68,Z 98.606,A -85,B 0,C 180,E1 -7084.968,E2 -7084.968} C_VEL
LIN {X 0,Y 481.638,Z 98.613,A -85,B 0,C 180,E1 -7087.967,E2 -7087.967} C_VEL
LIN {X 0,Y 480.961,Z 98.7,A -85,B 0,C 180,E1 -7088.433,E2 -7088.433} C_VEL
LIN {X 0,Y 478.143,Z 99.051,A -85,B 0,C 180,E1 -7089.161,E2 -7089.161} C_VEL
LIN {X 0,Y 475.317,Z 99.406,A -85,B 0,C 180,E1 -7089.898,E2 -7089.898} C_VEL
LIN {X 0,Y 474.646,Z 99.487,A -85,B 0,C 180,E1 -7090.373,E2 -7090.373} C_VEL
LIN {X 0,Y 474.686,Z 99.566,A -85,B 0,C 180,E1 -7091.662,E2 -7091.662} C_VEL
LIN {X 0,Y 476.876,Z 111.331,A -85,B 0,C 180,E1 -7093.959,E2 -7093.959} C_VEL
LIN {X 0,Y 476.547,Z 121.822,A -85,B 0,C 180,E1 -7095.848,E2 -7095.848} C_VEL
LIN {X 0,Y 479.998,Z 138.652,A -85,B 0,C 180,E1 -7096.25,E2 -7096.25} C_VEL
LIN {X 0,Y 478.918,Z 258.998,A -85,B 0,C 180,E1 -7098.091,E2 -7098.091} C_VEL
LIN {X 0,Y 478.598,Z 273.294,A -85,B 0,C 180,E1 -7098.486,E2 -7098.486} C_VEL
LIN {X 0,Y 478.216,Z 287.03,A -85,B 0,C 180,E1 -7099.04,E2 -7099.04} C_VEL
LIN {X 0,Y 477.645,Z 299.872,A -85,B 0,C 180,E1 -7099.723,E2 -7099.723} C_VEL
LIN {X 0,Y 477.012,Z 312.332,A -85,B 0,C 180,E1 -7100.566,E2 -7100.566} C_VEL
LIN {X 0,Y 476.413,Z 324.85,A -85,B 0,C 180,E1 -7101.624,E2 -7101.624} C_VEL
LIN {X 0,Y 475.851,Z 336.053,A -85,B 0,C 180,E1 -7102.788,E2 -7102.788} C_VEL
LIN {X 0,Y 475.23,Z 346.083,A -85,B 0,C 180,E1 -7104.058,E2 -7104.058} C_VEL
LIN {X 0,Y 474.743,Z 354.42,A -85,B 0,C 180,E1 -7105.33,E2 -7105.33} C_VEL
LIN {X 0,Y 474.346,Z 362.392,A -85,B 0,C 180,E1 -7106.815,E2 -7106.815} C_VEL
LIN {X 0,Y 473.954,Z 368.836,A -85,B 0,C 180,E1 -7108.301,E2 -7108.301} C_VEL
LIN {X 0,Y 473.935,Z 373.302,A -85,B 0,C 180,E1 -7109.575,E2 -7109.575} C_VEL
LIN {X 0,Y 473.76,Z 376.834,A -85,B 0,C 180,E1 -7110.85,E2 -7110.85} C_VEL
LIN {X 0,Y 473.763,Z 380.296,A -85,B 0,C 180,E1 -7112.551,E2 -7112.551} C_VEL
LIN {X 0,Y 473.694,Z 382.384,A -85,B 0,C 180,E1 -7114.254,E2 -7114.254} C_VEL
LIN {X 0,Y 473.746,Z 383.141,A -85,B 0,C 180,E1 -7115.961,E2 -7115.961} C_VEL
LIN {X 0,Y 473.715,Z 382.576,A -85,B 0,C 180,E1 -7117.673,E2 -7117.673} C_VEL
LIN {X 0,Y 473.679,Z 380.654,A -85,B 0,C 180,E1 -7119.393,E2 -7119.393} C_VEL
LIN {X 0,Y 473.865,Z 377.308,A -85,B 0,C 180,E1 -7121.117,E2 -7121.117} C_VEL
LIN {X 0,Y 473.97,Z 373.825,A -85,B 0,C 180,E1 -7122.416,E2 -7122.416} C_VEL
LIN {X 0,Y 474.108,Z 369.388,A -85,B 0,C 180,E1 -7123.72,E2 -7123.72} C_VEL
LIN {X 0,Y 474.383,Z 362.932,A -85,B 0,C 180,E1 -7125.246,E2 -7125.246} C_VEL
LIN {X 0,Y 474.833,Z 354.87,A -85,B 0,C 180,E1 -7126.775,E2 -7126.775} C_VEL
LIN {X 0,Y 475.311,Z 346.387,A -85,B 0,C 180,E1 -7128.09,E2 -7128.09} C_VEL
LIN {X 0,Y 475.928,Z 336.491,A -85,B 0,C 180,E1 -7129.361,E2 -7129.361} C_VEL
LIN {X 0,Y 476.531,Z 325.713,A -85,B 0,C 180,E1 -7130.504,E2 -7130.504} C_VEL
LIN {X 0,Y 477.129,Z 314.364,A -85,B 0,C 180,E1 -7131.494,E2 -7131.494} C_VEL
LIN {X 0,Y 477.785,Z 301.596,A -85,B 0,C 180,E1 -7132.393,E2 -7132.393} C_VEL
LIN {X 0,Y 478.432,Z 288.04,A -85,B 0,C 180,E1 -7133.138,E2 -7133.138} C_VEL
LIN {X 0,Y 478.868,Z 274.046,A -85,B 0,C 180,E1 -7133.717,E2 -7133.717} C_VEL
LIN {X 0,Y 479.199,Z 260.628,A -85,B 0,C 180,E1 -7134.102,E2 -7134.102} C_VEL
LIN {X 0,Y 479.503,Z 236.517,A -85,B 0,C 180,E1 -7134.506,E2 -7134.506} C_VEL
LIN {X 0,Y 480.464,Z 138.653,A -85,B 0,C 180,E1 -7135.999,E2 -7135.999} C_VEL
LIN {X 0,Y 476.762,Z 121.793,A -85,B 0,C 180,E1 -7136.453,E2 -7136.453} C_VEL
LIN {X 0,Y 477.136,Z 112.736,A -85,B 0,C 180,E1 -7138.122,E2 -7138.122} C_VEL
LIN {X 0,Y 475.732,Z 104.737,A -85,B 0,C 180,E1 -7139.723,E2 -7139.723} C_VEL
LIN {X 0,Y 474.562,Z 99.499,A -85,B 0,C 180,E1 -7140.848,E2 -7140.848} C_VEL
LIN {X 0,Y 474.609,Z 99.489,A -85,B 0,C 180,E1 -7143.223,E2 -7143.223} C_VEL
LIN {X 0,Y 474.568,Z 99.494,A -85,B 0,C 180,E1 -7146.325,E2 -7146.325} C_VEL
LIN {X 0,Y 474.599,Z 99.494,A -85,B 0,C 180,E1 -7149.55,E2 -7149.55} C_VEL
LIN {X 0,Y 474.566,Z 99.494,A -85,B 0,C 180,E1 -7152.94,E2 -7152.94} C_VEL
LIN {X 0,Y 474.602,Z 99.488,A -85,B 0,C 180,E1 -7155.894,E2 -7155.894} C_VEL
LIN {X 0,Y 474.592,Z 99.489,A -85,B 0,C 180,E1 -7159.339,E2 -7159.339} C_VEL
LIN {X 0,Y 474.593,Z 99.493,A -85,B 0,C 180,E1 -7161.707,E2 -7161.707} C_VEL
LIN {X 0,Y 474.619,Z 99.486,A -85,B 0,C 180,E1 -7164.725,E2 -7164.725} C_VEL
LIN {X 0,Y 474.636,Z 99.485,A -85,B 0,C 180,E1 -7167.787,E2 -7167.787} C_VEL
LIN {X 0,Y 474.6,Z 99.491,A -85,B 0,C 180,E1 -7170.89,E2 -7170.89} C_VEL
LIN {X 0,Y 474.583,Z 99.488,A -85,B 0,C 180,E1 -7173.624,E2 -7173.624} C_VEL
LIN {X 0,Y 474.635,Z 99.49,A -85,B 0,C 180,E1 -7176.642,E2 -7176.642} C_VEL
LIN {X 0,Y 474.653,Z 99.483,A -85,B 0,C 180,E1 -7180.089,E2 -7180.089} C_VEL
LIN {X 0,Y 474.635,Z 99.489,A -85,B 0,C 180,E1 -7182.774,E2 -7182.774} C_VEL
LIN {X 0,Y 474.638,Z 99.481,A -85,B 0,C 180,E1 -7185.42,E2 -7185.42} C_VEL
LIN {X 0,Y 474.705,Z 99.477,A -85,B 0,C 180,E1 -7188.037,E2 -7188.037} C_VEL
LIN {X 0,Y 474.712,Z 99.469,A -85,B 0,C 180,E1 -7191.486,E2 -7191.486} C_VEL
LIN {X 0,Y 474.745,Z 99.468,A -85,B 0,C 180,E1 -7194.904,E2 -7194.904} C_VEL
LIN {X 0,Y 474.887,Z 99.451,A -85,B 0,C 180,E1 -7197.455,E2 -7197.455} C_VEL
LIN {X 0,Y 474.912,Z 99.452,A -85,B 0,C 180,E1 -7200,E2 -7200} C_VEL
LIN {X 0,Y 474.887,Z 99.452,A -85,B 0,C 180,E1 -7202.545,E2 -7202.545} C_VEL
LIN {X 0,Y 474.751,Z 99.469,A -85,B 0,C 180,E1 -7205.948,E2 -7205.948} C_VEL
LIN {X 0,Y 474.713,Z 99.474,A -85,B 0,C 180,E1 -7208.514,E2 -7208.514} C_VEL
LIN {X 0,Y 474.705,Z 99.476,A -85,B 0,C 180,E1 -7211.962,E2 -7211.962} C_VEL
LIN {X 0,Y 474.7,Z 99.476,A -85,B 0,C 180,E1 -7215.456,E2 -7215.456} C_VEL
LIN {X 0,Y 474.666,Z 99.484,A -85,B 0,C 180,E1 -7219.01,E2 -7219.01} C_VEL
LIN {X 0,Y 474.589,Z 99.489,A -85,B 0,C 180,E1 -7221.729,E2 -7221.729} C_VEL
LIN {X 0,Y 474.658,Z 99.48,A -85,B 0,C 180,E1 -7224.493,E2 -7224.493} C_VEL
LIN {X 0,Y 474.682,Z 99.479,A -85,B 0,C 180,E1 -7227.334,E2 -7227.334} C_VEL
LIN {X 0,Y 474.606,Z 99.488,A -85,B 0,C 180,E1 -7230.23,E2 -7230.23} C_VEL
LIN {X 0,Y 474.644,Z 99.485,A -85,B 0,C 180,E1 -7233.22,E2 -7233.22} C_VEL
LIN {X 0,Y 474.59,Z 99.491,A -85,B 0,C 180,E1 -7236.323,E2 -7236.323} C_VEL
LIN {X 0,Y 474.618,Z 99.478,A -85,B 0,C 180,E1 -7239.646,E2 -7239.646} C_VEL
LIN {X 0,Y 474.615,Z 99.487,A -85,B 0,C 180,E1 -7242.934,E2 -7242.934} C_VEL
LIN {X 0,Y 474.607,Z 99.488,A -85,B 0,C 180,E1 -7245.895,E2 -7245.895} C_VEL
LIN {X 0,Y 474.629,Z 99.485,A -85,B 0,C 180,E1 -7249.041,E2 -7249.041} C_VEL
LIN {X 0,Y 474.611,Z 99.489,A -85,B 0,C 180,E1 -7251.704,E2 -7251.704} C_VEL
LIN {X 0,Y 474.625,Z 99.484,A -85,B 0,C 180,E1 -7254.726,E2 -7254.726} C_VEL
LIN {X 0,Y 474.637,Z 99.484,A -85,B 0,C 180,E1 -7257.788,E2 -7257.788} C_VEL
LIN {X 0,Y 474.625,Z 99.488,A -85,B 0,C 180,E1 -7260.884,E2 -7260.884} C_VEL
LIN {X 0,Y 474.684,Z 99.526,A -85,B 0,C 180,E1 -7262.431,E2 -7262.431} C_VEL
LIN {X 0,Y 477.706,Z 113.339,A -85,B 0,C 180,E1 -7264.978,E2 -7264.978} C_VEL
LIN {X 0,Y 477.789,Z 118.095,A -85,B 0,C 180,E1 -7265.781,E2 -7265.781} C_VEL
LIN {X 0,Y 476.718,Z 138.201,A -85,B 0,C 180,E1 -7269.053,E2 -7269.053} C_VEL
LIN {X 0,Y 476.538,Z 141.451,A -85,B 0,C 180,E1 -7269.575,E2 -7269.575} C_VEL
LIN {X 0,Y 480.206,Z 161.29,A -85,B 0,C 180,E1 -7270.071,E2 -7270.071} C_VEL
LIN {X 0,Y 479.251,Z 273.428,A -85,B 0,C 180,E1 -7271.788,E2 -7271.788} C_VEL
LIN {X 0,Y 478.875,Z 287.875,A -85,B 0,C 180,E1 -7272.105,E2 -7272.105} C_VEL
LIN {X 0,Y 478.419,Z 301.797,A -85,B 0,C 180,E1 -7272.584,E2 -7272.584} C_VEL
LIN {X 0,Y 477.915,Z 314.388,A -85,B 0,C 180,E1 -7273.176,E2 -7273.176} C_VEL
LIN {X 0,Y 477.251,Z 327.51,A -85,B 0,C 180,E1 -7273.972,E2 -7273.972} C_VEL
LIN {X 0,Y 476.549,Z 340.128,A -85,B 0,C 180,E1 -7274.934,E2 -7274.934} C_VEL
LIN {X 0,Y 475.892,Z 351.537,A -85,B 0,C 180,E1 -7276.005,E2 -7276.005} C_VEL
LIN {X 0,Y 475.36,Z 361.899,A -85,B 0,C 180,E1 -7277.187,E2 -7277.187} C_VEL
LIN {X 0,Y 474.874,Z 371.274,A -85,B 0,C 180,E1 -7278.475,E2 -7278.475} C_VEL
LIN {X 0,Y 474.356,Z 380.213,A -85,B 0,C 180,E1 -7279.974,E2 -7279.974} C_VEL
LIN {X 0,Y 474.079,Z 387.456,A -85,B 0,C 180,E1 -7281.475,E2 -7281.475} C_VEL
LIN {X 0,Y 473.889,Z 393.974,A -85,B 0,C 180,E1 -7283.186,E2 -7283.186} C_VEL
LIN {X 0,Y 473.816,Z 398.853,A -85,B 0,C 180,E1 -7284.894,E2 -7284.894} C_VEL
LIN {X 0,Y 473.755,Z 402.244,A -85,B 0,C 180,E1 -7286.598,E2 -7286.598} C_VEL
LIN {X 0,Y 473.695,Z 404.244,A -85,B 0,C 180,E1 -7288.299,E2 -7288.299} C_VEL
LIN {X 0,Y 473.669,Z 404.896,A -85,B 0,C 180,E1 -7290,E2 -7290} C_VEL
LIN {X 0,Y 473.695,Z 404.211,A -85,B 0,C 180,E1 -7291.7,E2 -7291.7} C_VEL
LIN {X 0,Y 473.754,Z 402.18,A -85,B 0,C 180,E1 -7293.402,E2 -7293.402} C_VEL
LIN {X 0,Y 473.816,Z 398.746,A -85,B 0,C 180,E1 -7295.106,E2 -7295.106} C_VEL
LIN {X 0,Y 473.888,Z 393.804,A -85,B 0,C 180,E1 -7296.814,E2 -7296.814} C_VEL
LIN {X 0,Y 474.077,Z 387.21,A -85,B 0,C 180,E1 -7298.525,E2 -7298.525} C_VEL
LIN {X 0,Y 474.341,Z 379.867,A -85,B 0,C 180,E1 -7300.026,E2 -7300.026} C_VEL
LIN {X 0,Y 474.836,Z 370.749,A -85,B 0,C 180,E1 -7301.526,E2 -7301.526} C_VEL
LIN {X 0,Y 475.269,Z 361.181,A -85,B 0,C 180,E1 -7302.815,E2 -7302.815} C_VEL
LIN {X 0,Y 475.853,Z 350.58,A -85,B 0,C 180,E1 -7303.995,E2 -7303.995} C_VEL
LIN {X 0,Y 476.427,Z 338.859,A -85,B 0,C 180,E1 -7305.07,E2 -7305.07} C_VEL
LIN {X 0,Y 477.05,Z 327.419,A -85,B 0,C 180,E1 -7305.925,E2 -7305.925} C_VEL
LIN {X 0,Y 477.687,Z 314.42,A -85,B 0,C 180,E1 -7306.705,E2 -7306.705} C_VEL
LIN {X 0,Y 478.175,Z 300.622,A -85,B 0,C 180,E1 -7307.342,E2 -7307.342} C_VEL
LIN {X 0,Y 478.648,Z 286.517,A -85,B 0,C 180,E1 -7307.807,E2 -7307.807} C_VEL
LIN {X 0,Y 478.942,Z 271.58,A -85,B 0,C 180,E1 -7308.114,E2 -7308.114} C_VEL
LIN {X 0,Y 479.847,Z 161.509,A -85,B 0,C 180,E1 -7309.775,E2 -7309.775} C_VEL
LIN {X 0,Y 476.356,Z 141.557,A -85,B 0,C 180,E1 -7310.23,E2 -7310.23} C_VEL
LIN {X 0,Y 477.294,Z 120.382,A -85,B 0,C 180,E1 -7313.605,E2 -7313.605} C_VEL
LIN {X 0,Y 477.491,Z 113.001,A -85,B 0,C 180,E1 -7314.802,E2 -7314.802} C_VEL
LIN {X 0,Y 474.718,Z 99.477,A -85,B 0,C 180,E1 -7317.208,E2 -7317.208} C_VEL
LIN {X 0,Y 474.606,Z 99.495,A -85,B 0,C 180,E1 -7320.23,E2 -7320.23} C_VEL
LIN {X 0,Y 474.643,Z 99.482,A -85,B 0,C 180,E1 -7323.22,E2 -7323.22} C_VEL
LIN {X 0,Y 474.588,Z 99.494,A -85,B 0,C 180,E1 -7326.323,E2 -7326.323} C_VEL
LIN {X 0,Y 474.627,Z 99.488,A -85,B 0,C 180,E1 -7329.647,E2 -7329.647} C_VEL
LIN {X 0,Y 474.614,Z 99.486,A -85,B 0,C 180,E1 -7332.934,E2 -7332.934} C_VEL
LIN {X 0,Y 474.618,Z 99.491,A -85,B 0,C 180,E1 -7335.896,E2 -7335.896} C_VEL
LIN {X 0,Y 474.631,Z 99.485,A -85,B 0,C 180,E1 -7339.04,E2 -7339.04} C_VEL
LIN {X 0,Y 474.608,Z 99.493,A -85,B 0,C 180,E1 -7341.704,E2 -7341.704} C_VEL
LIN {X 0,Y 474.623,Z 99.485,A -85,B 0,C 180,E1 -7344.726,E2 -7344.726} C_VEL
LIN {X 0,Y 474.635,Z 99.486,A -85,B 0,C 180,E1 -7347.788,E2 -7347.788} C_VEL
LIN {X 0,Y 474.623,Z 99.488,A -85,B 0,C 180,E1 -7350.884,E2 -7350.884} C_VEL
LIN {X 0,Y 474.659,Z 99.482,A -85,B 0,C 180,E1 -7353.628,E2 -7353.628} C_VEL
LIN {X 0,Y 474.634,Z 99.486,A -85,B 0,C 180,E1 -7356.641,E2 -7356.641} C_VEL
LIN {X 0,Y 474.653,Z 99.481,A -85,B 0,C 180,E1 -7360.09,E2 -7360.09} C_VEL
LIN {X 0,Y 474.647,Z 99.488,A -85,B 0,C 180,E1 -7362.774,E2 -7362.774} C_VEL
LIN {X 0,Y 474.647,Z 99.483,A -85,B 0,C 180,E1 -7365.421,E2 -7365.421} C_VEL
LIN {X 0,Y 474.703,Z 99.475,A -85,B 0,C 180,E1 -7368.038,E2 -7368.038} C_VEL
LIN {X 0,Y 474.727,Z 99.472,A -85,B 0,C 180,E1 -7371.487,E2 -7371.487} C_VEL
LIN {X 0,Y 474.771,Z 99.468,A -85,B 0,C 180,E1 -7374.052,E2 -7374.052} C_VEL
LIN {X 0,Y 474.893,Z 99.451,A -85,B 0,C 180,E1 -7377.456,E2 -7377.456} C_VEL
LIN {X 0,Y 474.911,Z 99.453,A -85,B 0,C 180,E1 -7380,E2 -7380} C_VEL
LIN {X 0,Y 474.892,Z 99.455,A -85,B 0,C 180,E1 -7382.545,E2 -7382.545} C_VEL
LIN {X 0,Y 474.757,Z 99.474,A -85,B 0,C 180,E1 -7385.948,E2 -7385.948} C_VEL
LIN {X 0,Y 474.727,Z 99.474,A -85,B 0,C 180,E1 -7388.514,E2 -7388.514} C_VEL
LIN {X 0,Y 474.704,Z 99.482,A -85,B 0,C 180,E1 -7391.963,E2 -7391.963} C_VEL
LIN {X 0,Y 474.699,Z 99.479,A -85,B 0,C 180,E1 -7395.456,E2 -7395.456} C_VEL
LIN {X 0,Y 474.661,Z 99.481,A -85,B 0,C 180,E1 -7399.011,E2 -7399.011} C_VEL
LIN {X 0,Y 474.588,Z 99.495,A -85,B 0,C 180,E1 -7401.729,E2 -7401.729} C_VEL
LIN {X 0,Y 474.64,Z 99.482,A -85,B 0,C 180,E1 -7404.494,E2 -7404.494} C_VEL
LIN {X 0,Y 474.681,Z 99.485,A -85,B 0,C 180,E1 -7407.335,E2 -7407.335} C_VEL
LIN {X 0,Y 474.603,Z 99.489,A -85,B 0,C 180,E1 -7410.81,E2 -7410.81} C_VEL
LIN {X 0,Y 474.625,Z 99.492,A -85,B 0,C 180,E1 -7413.222,E2 -7413.222} C_VEL
LIN {X 0,Y 474.588,Z 99.489,A -85,B 0,C 180,E1 -7416.324,E2 -7416.324} C_VEL
LIN {X 0,Y 474.616,Z 99.486,A -85,B 0,C 180,E1 -7419.646,E2 -7419.646} C_VEL
LIN {X 0,Y 474.624,Z 99.485,A -85,B 0,C 180,E1 -7422.237,E2 -7422.237} C_VEL
LIN {X 0,Y 474.617,Z 99.487,A -85,B 0,C 180,E1 -7425.298,E2 -7425.298} C_VEL
LIN {X 0,Y 474.616,Z 99.487,A -85,B 0,C 180,E1 -7428.214,E2 -7428.214} C_VEL
LIN {X 0,Y 474.611,Z 99.486,A -85,B 0,C 180,E1 -7431.543,E2 -7431.543} C_VEL
LIN {X 0,Y 474.623,Z 99.489,A -85,B 0,C 180,E1 -7434.726,E2 -7434.726} C_VEL
LIN {X 0,Y 474.637,Z 99.484,A -85,B 0,C 180,E1 -7437.788,E2 -7437.788} C_VEL
LIN {X 0,Y 474.608,Z 99.488,A -85,B 0,C 180,E1 -7440.889,E2 -7440.889} C_VEL
LIN {X 0,Y 474.606,Z 99.488,A -85,B 0,C 180,E1 -7443.625,E2 -7443.625} C_VEL
LIN {X 0,Y 474.637,Z 99.484,A -85,B 0,C 180,E1 -7446.642,E2 -7446.642} C_VEL
LIN {X 0,Y 474.656,Z 99.488,A -85,B 0,C 180,E1 -7450.09,E2 -7450.09} C_VEL
LIN {X 0,Y 474.646,Z 99.487,A -85,B 0,C 180,E1 -7450.373,E2 -7450.373} C_VEL
LIN {X 0,Y 474.405,Z 99.828,A -85,B 0,C 180,E1 -7450.841,E2 -7450.841} C_VEL
LIN {X 0,Y 473.417,Z 101.378,A -85,B 0,C 180,E1 -7451.517,E2 -7451.517} C_VEL
LIN {X 0,Y 472.087,Z 103.798,A -85,B 0,C 180,E1 -7452.153,E2 -7452.153} C_VEL
LIN {X 0,Y 470.433,Z 107.913,A -85,B 0,C 180,E1 -7452.98,E2 -7452.98} C_VEL
LIN {X 0,Y 469.89,Z 112.337,A -85,B 0,C 180,E1 -7453.801,E2 -7453.801} C_VEL
LIN {X 0,Y 469.61,Z 121.96,A -85,B 0,C 180,E1 -7455.562,E2 -7455.562} C_VEL
LIN {X 0,Y 473.245,Z 139.623,A -85,B 0,C 180,E1 -7455.992,E2 -7455.992} C_VEL
LIN {X 0,Y 472.145,Z 258.707,A -85,B 0,C 180,E1 -7457.836,E2 -7457.836} C_VEL
LIN {X 0,Y 471.811,Z 273.158,A -85,B 0,C 180,E1 -7458.236,E2 -7458.236} C_VEL
LIN {X 0,Y 471.387,Z 287.533,A -85,B 0,C 180,E1 -7458.824,E2 -7458.824} C_VEL
LIN {X 0,Y 470.74,Z 301.179,A -85,B 0,C 180,E1 -7459.571,E2 -7459.571} C_VEL
LIN {X 0,Y 470.079,Z 313.423,A -85,B 0,C 180,E1 -7460.426,E2 -7460.426} C_VEL
LIN {X 0,Y 469.464,Z 325.777,A -85,B 0,C 180,E1 -7461.499,E2 -7461.499} C_VEL
LIN {X 0,Y 468.848,Z 336.817,A -85,B 0,C 180,E1 -7462.68,E2 -7462.68} C_VEL
LIN {X 0,Y 468.21,Z 346.74,A -85,B 0,C 180,E1 -7463.969,E2 -7463.969} C_VEL
LIN {X 0,Y 467.698,Z 354.995,A -85,B 0,C 180,E1 -7465.259,E2 -7465.259} C_VEL
LIN {X 0,Y 467.242,Z 361.902,A -85,B 0,C 180,E1 -7466.551,E2 -7466.551} C_VEL
LIN {X 0,Y 467.108,Z 367.596,A -85,B 0,C 180,E1 -7467.844,E2 -7467.844} C_VEL
LIN {X 0,Y 466.779,Z 372.304,A -85,B 0,C 180,E1 -7469.137,E2 -7469.137} C_VEL
LIN {X 0,Y 466.736,Z 376.121,A -85,B 0,C 180,E1 -7470.432,E2 -7470.432} C_VEL
LIN {X 0,Y 466.677,Z 379.058,A -85,B 0,C 180,E1 -7471.726,E2 -7471.726} C_VEL
LIN {X 0,Y 466.68,Z 381.766,A -85,B 0,C 180,E1 -7473.454,E2 -7473.454} C_VEL
LIN {X 0,Y 466.652,Z 383.132,A -85,B 0,C 180,E1 -7475.185,E2 -7475.185} C_VEL
LIN {X 0,Y 466.68,Z 383.168,A -85,B 0,C 180,E1 -7476.92,E2 -7476.92} C_VEL
LIN {X 0,Y 466.588,Z 381.862,A -85,B 0,C 180,E1 -7478.663,E2 -7478.663} C_VEL
LIN {X 0,Y 466.689,Z 379.172,A -85,B 0,C 180,E1 -7480.411,E2 -7480.411} C_VEL
LIN {X 0,Y 466.872,Z 375.023,A -85,B 0,C 180,E1 -7482.166,E2 -7482.166} C_VEL
LIN {X 0,Y 467.064,Z 369.273,A -85,B 0,C 180,E1 -7483.931,E2 -7483.931} C_VEL
LIN {X 0,Y 467.395,Z 362.75,A -85,B 0,C 180,E1 -7485.48,E2 -7485.48} C_VEL
LIN {X 0,Y 467.87,Z 354.613,A -85,B 0,C 180,E1 -7487.033,E2 -7487.033} C_VEL
LIN {X 0,Y 468.396,Z 346.047,A -85,B 0,C 180,E1 -7488.366,E2 -7488.366} C_VEL
LIN {X 0,Y 469.055,Z 335.627,A -85,B 0,C 180,E1 -7489.702,E2 -7489.702} C_VEL
LIN {X 0,Y 469.707,Z 325.091,A -85,B 0,C 180,E1 -7490.816,E2 -7490.816} C_VEL
LIN {X 0,Y 470.378,Z 313.576,A -85,B 0,C 180,E1 -7491.818,E2 -7491.818} C_VEL
LIN {X 0,Y 471.064,Z 300.654,A -85,B 0,C 180,E1 -7492.725,E2 -7492.725} C_VEL
LIN {X 0,Y 471.779,Z 286.712,A -85,B 0,C 180,E1 -7493.484,E2 -7493.484} C_VEL
LIN {X 0,Y 472.237,Z 272.985,A -85,B 0,C 180,E1 -7494.042,E2 -7494.042} C_VEL
LIN {X 0,Y 472.621,Z 258.98,A -85,B 0,C 180,E1 -7494.43,E2 -7494.43} C_VEL
LIN {X 0,Y 473.796,Z 139.407,A -85,B 0,C 180,E1 -7496.307,E2 -7496.307} C_VEL
LIN {X 0,Y 469.919,Z 121.856,A -85,B 0,C 180,E1 -7496.809,E2 -7496.809} C_VEL
LIN {X 0,Y 470.218,Z 113.939,A -85,B 0,C 180,E1 -7498.293,E2 -7498.293} C_VEL
LIN {X 0,Y 468.52,Z 104.775,A -85,B 0,C 180,E1 -7500.166,E2 -7500.166} C_VEL
LIN {X 0,Y 467.531,Z 100.375,A -85,B 0,C 180,E1 -7501.099,E2 -7501.099} C_VEL
LIN {X 0,Y 467.563,Z 100.369,A -85,B 0,C 180,E1 -7504.237,E2 -7504.237} C_VEL
LIN {X 0,Y 467.514,Z 100.37,A -85,B 0,C 180,E1 -7507.18,E2 -7507.18} C_VEL
LIN {X 0,Y 467.518,Z 100.374,A -85,B 0,C 180,E1 -7510.271,E2 -7510.271} C_VEL
LIN {X 0,Y 467.517,Z 100.372,A -85,B 0,C 180,E1 -7512.568,E2 -7512.568} C_VEL
LIN {X 0,Y 467.565,Z 100.367,A -85,B 0,C 180,E1 -7515.052,E2 -7515.052} C_VEL
LIN {X 0,Y 467.561,Z 100.366,A -85,B 0,C 180,E1 -7518.726,E2 -7518.726} C_VEL
LIN {X 0,Y 467.544,Z 100.369,A -85,B 0,C 180,E1 -7521.953,E2 -7521.953} C_VEL
LIN {X 0,Y 467.557,Z 100.371,A -85,B 0,C 180,E1 -7525.166,E2 -7525.166} C_VEL
LIN {X 0,Y 467.582,Z 100.363,A -85,B 0,C 180,E1 -7528.26,E2 -7528.26} C_VEL
LIN {X 0,Y 467.546,Z 100.372,A -85,B 0,C 180,E1 -7531.248,E2 -7531.248} C_VEL
LIN {X 0,Y 467.577,Z 100.362,A -85,B 0,C 180,E1 -7534.401,E2 -7534.401} C_VEL
LIN {X 0,Y 467.573,Z 100.364,A -85,B 0,C 180,E1 -7536.995,E2 -7536.995} C_VEL
LIN {X 0,Y 467.622,Z 100.358,A -85,B 0,C 180,E1 -7539.777,E2 -7539.777} C_VEL
LIN {X 0,Y 467.596,Z 100.362,A -85,B 0,C 180,E1 -7542.506,E2 -7542.506} C_VEL
LIN {X 0,Y 467.598,Z 100.359,A -85,B 0,C 180,E1 -7545.196,E2 -7545.196} C_VEL
LIN {X 0,Y 467.657,Z 100.353,A -85,B 0,C 180,E1 -7547.854,E2 -7547.854} C_VEL
LIN {X 0,Y 467.67,Z 100.345,A -85,B 0,C 180,E1 -7551.357,E2 -7551.357} C_VEL
LIN {X 0,Y 467.721,Z 100.35,A -85,B 0,C 180,E1 -7553.962,E2 -7553.962} C_VEL
LIN {X 0,Y 467.852,Z 100.327,A -85,B 0,C 180,E1 -7557.417,E2 -7557.417} C_VEL
LIN {X 0,Y 467.882,Z 100.328,A -85,B 0,C 180,E1 -7560,E2 -7560} C_VEL
LIN {X 0,Y 467.852,Z 100.328,A -85,B 0,C 180,E1 -7562.583,E2 -7562.583} C_VEL
LIN {X 0,Y 467.714,Z 100.344,A -85,B 0,C 180,E1 -7566.038,E2 -7566.038} C_VEL
LIN {X 0,Y 467.671,Z 100.351,A -85,B 0,C 180,E1 -7568.643,E2 -7568.643} C_VEL
LIN {X 0,Y 467.657,Z 100.352,A -85,B 0,C 180,E1 -7572.145,E2 -7572.145} C_VEL
LIN {X 0,Y 467.64,Z 100.352,A -85,B 0,C 180,E1 -7575.695,E2 -7575.695} C_VEL
LIN {X 0,Y 467.618,Z 100.359,A -85,B 0,C 180,E1 -7578.764,E2 -7578.764} C_VEL
LIN {X 0,Y 467.581,Z 100.364,A -85,B 0,C 180,E1 -7581.268,E2 -7581.268} C_VEL
LIN {X 0,Y 467.572,Z 100.361,A -85,B 0,C 180,E1 -7583.943,E2 -7583.943} C_VEL
LIN {X 0,Y 467.617,Z 100.362,A -85,B 0,C 180,E1 -7586.8,E2 -7586.8} C_VEL
LIN {X 0,Y 467.555,Z 100.365,A -85,B 0,C 180,E1 -7589.738,E2 -7589.738} C_VEL
LIN {X 0,Y 467.584,Z 100.366,A -85,B 0,C 180,E1 -7592.758,E2 -7592.758} C_VEL
LIN {X 0,Y 467.554,Z 100.364,A -85,B 0,C 180,E1 -7595.89,E2 -7595.89} C_VEL
LIN {X 0,Y 467.56,Z 100.358,A -85,B 0,C 180,E1 -7599.147,E2 -7599.147} C_VEL
LIN {X 0,Y 467.587,Z 100.366,A -85,B 0,C 180,E1 -7602.567,E2 -7602.567} C_VEL
LIN {X 0,Y 467.567,Z 100.362,A -85,B 0,C 180,E1 -7605.053,E2 -7605.053} C_VEL
